# B&R Automation Studio project Panasonic_LinkaPowerCP2_A2021055 (part 8)

#### SKTcpClientTrace.c - SKTcpClientTrace
```c
/*************************************************************
*
*         projekt: SKTcp - Panasonic
*
*         autor: Ing. Milan Jun
*         company: B+R Automatizace spol. s r.o.
*         date: 10.09.2020
*
*/

#include <bur/plctypes.h>
#ifdef __cplusplus
	extern "C"
	{
#endif
#include "SKTcp.h"
#ifdef __cplusplus
	};
#endif

/* SKTcpClientTrace */
void SKTcpClientTrace(struct SKTcpClientTrace* inst)
{

	if( inst->Enable == 1 ) {

		if(( inst->Cmd.Send == 1 ) && ( inst->Internal.SendOld == 0 )) {
			inst->Internal.cmdSend = 1 ;
		}
		inst->Internal.SendOld = inst->Cmd.Send ;

		if(( inst->Cmd.Close == 1 ) && ( inst->Internal.CloseOld == 0 )) {
			inst->Internal.cmdClose = 1 ;
		} else {
			if( inst->Cmd.Close == 0 ) {
				inst->Internal.cmdClose = 0 ;
			}
		}
		inst->Internal.CloseOld = inst->Cmd.Close ;

		inst->Status.staSending = 0 ;
		inst->Status.staReceiving = 0 ;
		inst->Status.staReadyToSend = 0 ;
		inst->Status.staReadyToClose = 0 ;

		switch( inst->Internal.Step ) {

			case 0:
				inst->Status.staReadyToSend = 1 ;
				inst->Status.staSending = 0;
				inst->Internal.TimerIddle.IN = 0;

				if( inst->Internal.cmdSend == 1 ) {
					inst->FBStatus = 0xFFFF ;
					inst->Status.staSent = 0 ;
					inst->Status.staReceived = 0 ;

					inst->Status.staError = 0 ;
					inst->Status.staErrorSent = 0 ;
					inst->Status.staErrorOpen = 0 ;
					inst->Status.staErrorRecv = 0 ;
					inst->Status.staErrorRecvTout = 0 ;
					inst->Status.staErrorOpen = 0 ;
					inst->Status.staErrorIoctl = 0 ;
					inst->Status.staErrorClient = 0 ;
					inst->Status.staErrorConn = 0 ;
					inst->Status.staErrorConnTout = 0 ;

					inst->Status.RecvSize = 0 ;
					brsmemset((void*)&inst->Status.DataRecv[0], 0, sizeof(inst->Status.DataRecv)) ;

					inst->Internal.TimerConn.IN = 1 ;
					inst->Internal.TimerConn.PT = inst->Params.ConnTimeout ;

					inst->Internal.TCP_Open.enable = 1;
					inst->Internal.TCP_Open.pIfAddr = 0;
					inst->Internal.TCP_Open.port = inst->Params.IPportClient;
					inst->Internal.TCP_Open.options = 0;
					TcpOpen(&inst->Internal.TCP_Open);

					if( inst->Internal.TCP_Open.status == 0 ) {
						inst->Internal.Step = 4;
					}
					else if( inst->Internal.TimerConn.Q == 1 ) {
						inst->Internal.cmdSend = 0 ;
						inst->Status.staErrorOpen = 1 ;
						inst->Status.staErrorConn = 1 ;
						inst->Status.staErrorConnTout = 1 ;
						inst->Internal.Step = 99;
					} else if( inst->Internal.TCP_Open.status == ERR_FUB_BUSY ) {

					} else {
						if( inst->Internal.TCP_Open.status == tcpERR_ALREADY_EXIST ) {
							inst->Status.staErrorOpen = 1 ;
							inst->Internal.Step = 90;
						} else {
							inst->Status.staErrorOpen = 1 ;
							inst->Internal.Step = 99;
						}
						inst->Internal.cmdSend = 0 ;
					}
				}

				else if( inst->Cmd.Close == 1 ) {
					inst->Cmd.Close = 0 ;
					inst->Internal.Step = 40 ;
				}
				break ;

			case 4:
				inst->Internal.TimerIddle.IN = 1;
				inst->Internal.TimerIddle.PT = 1000;

				if( inst->Internal.TimerIddle.Q == 1 )
				{
					inst->Internal.TimerIddle.IN = 0 ;
					inst->Internal.Step = 5;
				}
				break ;

			case 5:
				inst->Internal.linger_opt.lLinger = 0;
				inst->Internal.linger_opt.lOnOff = 1;

				inst->Internal.TCP_Ioctl.enable = 1;
				inst->Internal.TCP_Ioctl.ident = inst->Internal.TCP_Open.ident;
				inst->Internal.TCP_Ioctl.ioctl = tcpSO_LINGER_SET;
				inst->Internal.TCP_Ioctl.pData = (UDINT)&(inst->Internal.linger_opt);
				inst->Internal.TCP_Ioctl.datalen = sizeof(inst->Internal.linger_opt);
				TcpIoctl(&inst->Internal.TCP_Ioctl);

				if( inst->Internal.TCP_Ioctl.status == 0 ) {
					inst->Internal.Step = 10;
				} else if( inst->Internal.TimerConn.Q == 1 ) {
					inst->Status.staErrorOpen = 1 ;
					inst->Status.staErrorConn = 1 ;
					inst->Status.staErrorConnTout = 1 ;
					inst->Internal.Step = 99;
				} else if( inst->Internal.TCP_Ioctl.status == ERR_FUB_BUSY ) {
				} else {
					inst->Status.staErrorIoctl = 1 ;
					inst->Internal.Step = 90;
				}
				break ;

			case 10:
				inst->Internal.TCP_Client.enable = 1;
				inst->Internal.TCP_Client.ident = inst->Internal.TCP_Open.ident ;
				inst->Internal.TCP_Client.portserv = inst->Params.IPportServ ;
				inst->Internal.TCP_Client.pServer = (UDINT)&inst->Params.IPaddrServ[0];
				TcpClient(&inst->Internal.TCP_Client) ;

				if( inst->Internal.TCP_Client.status == 0 ) {
					inst->Internal.Step = 15;
				} else if( inst->Internal.TimerConn.Q == 1 ) {
					inst->Status.staErrorOpen = 1 ;
					inst->Status.staErrorConn = 1 ;
					inst->Status.staErrorConnTout = 1 ;
					inst->Internal.Step = 90;
				} else if( inst->Internal.TCP_Client.status == ERR_FUB_BUSY ) {
				} else if( inst->Internal.TCP_Client.status == tcpERR_INVALID ) {
					inst->Status.staErrorClient = 1 ;
					inst->Status.staErrorConn = 1 ;
					inst->Internal.Step = 90;
				} else {
					inst->Status.staErrorClient = 1 ;
					inst->Internal.Step = 90;
				}
				break ;

			case 15:
				inst->Status.staReadyToSend = 1;
				inst->Status.staSending = 0;

				if ( inst->Internal.cmdSend == 1 ) {
					inst->Status.RecvSize = 0 ;
					inst->Internal.TimerRecv.IN = 0 ;
					inst->Internal.cmdSend = 0 ;
					brsmemset((void*)&inst->Status.DataRecv, 0, sizeof(inst->Status.DataRecv)) ;

					brsmemset((void*)&inst->Internal.Splitter.out, 0, sizeof(inst->Internal.Splitter.out));
					inst->Internal.Step = 18;
				}
				else if ( inst->Internal.cmdClose == 1 ) {
					inst->Internal.cmdClose=0;
					inst->Internal.Step = 40;
				}
				break ;

			case 18:

				inst->Status.staSending = 1;

				inst->Internal.oneskorenie.IN = 1;
				inst->Internal.oneskorenie.PT = 100; //ms  1000

				if ( inst->Internal.oneskorenie.Q == 1 ) {
					inst->Internal.oneskorenie.IN = 0;
					inst->Internal.Step = 19;
				}

				TON(&inst->Internal.oneskorenie);

				break ;

			case 19:

				inst->Params.Packet.internal.start = 0x02;
				inst->Params.Packet.internal.length_int = 0;
				//inst->Params.Packet.internal.xor = 0;
				inst->Params.Packet.internal.stop = 0x03;

				brsmemset((UDINT)&(inst->Params.Packet.internal.length_str), 0, sizeof(inst->Params.Packet.internal.length_str));
				brsmemset((UDINT)&(inst->Params.Packet.internal.xor_str), 0, sizeof(inst->Params.Packet.internal.xor_str));

				brsmemset((UDINT)&(inst->DataSend.send_data_a), 0, sizeof(inst->DataSend.send_data_a));
				brsstrcat((UDINT)&(inst->DataSend.send_data_a), (UDINT)&(inst->Params.Packet.type));
				brsstrcat((UDINT)&(inst->DataSend.send_data_a), (UDINT)&("|"));
				brsstrcat((UDINT)&(inst->DataSend.send_data_a), (UDINT)&(inst->Params.Packet.workplace));
				brsstrcat((UDINT)&(inst->DataSend.send_data_a), (UDINT)&("|"));
				brsstrcat((UDINT)&(inst->DataSend.send_data_a), (UDINT)&(inst->Params.Packet.rfid));
				brsstrcat((UDINT)&(inst->DataSend.send_data_a), (UDINT)&("|"));
				brsstrcat((UDINT)&(inst->DataSend.send_data_a), (UDINT)&(inst->Params.Packet.master));
				brsstrcat((UDINT)&(inst->DataSend.send_data_a), (UDINT)&("|"));
				brsstrcat((UDINT)&(inst->DataSend.send_data_a), (UDINT)&(inst->Params.Packet.dps1));
				brsstrcat((UDINT)&(inst->DataSend.send_data_a), (UDINT)&("|"));
				brsstrcat((UDINT)&(inst->DataSend.send_data_a), (UDINT)&(inst->Params.Packet.dps2));
				brsstrcat((UDINT)&(inst->DataSend.send_data_a), (UDINT)&("|"));
				brsstrcat((UDINT)&(inst->DataSend.send_data_a), (UDINT)&(inst->Params.Packet.dps3));
				brsstrcat((UDINT)&(inst->DataSend.send_data_a), (UDINT)&("|"));
				brsstrcat((UDINT)&(inst->DataSend.send_data_a), (UDINT)&(inst->Params.Packet.dps4));
				brsstrcat((UDINT)&(inst->DataSend.send_data_a), (UDINT)&("|"));
				brsstrcat((UDINT)&(inst->DataSend.send_data_a), (UDINT)&(inst->Params.Packet.dps5));
				brsstrcat((UDINT)&(inst->DataSend.send_data_a), (UDINT)&("|"));
				brsstrcat((UDINT)&(inst->DataSend.send_data_a), (UDINT)&(inst->Params.Packet.operator_id));
				brsstrcat((UDINT)&(inst->DataSend.send_data_a), (UDINT)&("|"));
				brsstrcat((UDINT)&(inst->DataSend.send_data_a), (UDINT)&(inst->Params.Packet.data_report));
				brsstrcat((UDINT)&(inst->DataSend.send_data_a), (UDINT)&("|"));
				brsstrcat((UDINT)&(inst->DataSend.send_data_a), (UDINT)&(inst->Params.Packet.result));

				inst->Params.Packet.internal.length_int = brsstrlen((UDINT)&inst->DataSend.send_data_a);

				inst->Params.Packet.internal.length_b_int = inst->Params.Packet.internal.length_int + SKTcpClientNod(inst->Params.Packet.internal.length_int);

				brsitoa(inst->Params.Packet.internal.length_b_int,(UDINT)&(inst->Params.Packet.internal.length_str));

				brsmemset((UDINT)&(inst->DataSend.send_data_b), 0, sizeof(inst->DataSend.send_data_b));
				brsstrcat((UDINT)&(inst->DataSend.send_data_b), (UDINT)&(inst->Params.Packet.internal.length_str));
				brsstrcat((UDINT)&(inst->DataSend.send_data_b), (UDINT)&("|"));
				brsstrcat((UDINT)&(inst->DataSend.send_data_b), (UDINT)&(inst->Params.Packet.type));
				brsstrcat((UDINT)&(inst->DataSend.send_data_b), (UDINT)&("|"));
				brsstrcat((UDINT)&(inst->DataSend.send_data_b), (UDINT)&(inst->Params.Packet.workplace));
				brsstrcat((UDINT)&(inst->DataSend.send_data_b), (UDINT)&("|"));
				brsstrcat((UDINT)&(inst->DataSend.send_data_b), (UDINT)&(inst->Params.Packet.rfid));
				brsstrcat((UDINT)&(inst->DataSend.send_data_b), (UDINT)&("|"));
				brsstrcat((UDINT)&(inst->DataSend.send_data_b), (UDINT)&(inst->Params.Packet.master));
				brsstrcat((UDINT)&(inst->DataSend.send_data_b), (UDINT)&("|"));
				brsstrcat((UDINT)&(inst->DataSend.send_data_b), (UDINT)&(inst->Params.Packet.dps1));
				brsstrcat((UDINT)&(inst->DataSend.send_data_b), (UDINT)&("|"));
				brsstrcat((UDINT)&(inst->DataSend.send_data_b), (UDINT)&(inst->Params.Packet.dps2));
				brsstrcat((UDINT)&(inst->DataSend.send_data_b), (UDINT)&("|"));
				brsstrcat((UDINT)&(inst->DataSend.send_data_b), (UDINT)&(inst->Params.Packet.dps3));
				brsstrcat((UDINT)&(inst->DataSend.send_data_b), (UDINT)&("|"));
				brsstrcat((UDINT)&(inst->DataSend.send_data_b), (UDINT)&(inst->Params.Packet.dps4));
				brsstrcat((UDINT)&(inst->DataSend.send_data_b), (UDINT)&("|"));
				brsstrcat((UDINT)&(inst->DataSend.send_data_b), (UDINT)&(inst->Params.Packet.dps5));
				brsstrcat((UDINT)&(inst->DataSend.send_data_b), (UDINT)&("|"));
				brsstrcat((UDINT)&(inst->DataSend.send_data_b), (UDINT)&(inst->Params.Packet.operator_id));
				brsstrcat((UDINT)&(inst->DataSend.send_data_b), (UDINT)&("|"));
				brsstrcat((UDINT)&(inst->DataSend.send_data_b), (UDINT)&(inst->Params.Packet.data_report));
				brsstrcat((UDINT)&(inst->DataSend.send_data_b), (UDINT)&("|"));
				brsstrcat((UDINT)&(inst->DataSend.send_data_b), (UDINT)&(inst->Params.Packet.result));
				brsstrcat((UDINT)&(inst->DataSend.send_data_b), (UDINT)&("|"));

				//inst->Params.Packet.internal.xor_str = SKTcpClientXor(inst->DataSend.send_data_b,inst->Params.Packet.internal.length_int);

				//SKTcpClientNod(inst->Params.Packet.internal.length_int);
				inst->Params.Packet.internal.xor_str = SKTcpClientXor(inst->DataSend.send_data_b, inst->Params.Packet.internal.length_b_int+2);

				brsmemset((UDINT)&(inst->DataSend.DataSend), 0, sizeof(inst->DataSend.DataSend));
				inst->DataSend.DataSend[0] = inst->Params.Packet.internal.start;
				brsstrcat((UDINT)&(inst->DataSend.DataSend), (UDINT)&(inst->Params.Packet.internal.length_str));
				brsstrcat((UDINT)&(inst->DataSend.DataSend), (UDINT)&("|"));
				brsstrcat((UDINT)&(inst->DataSend.DataSend), (UDINT)&(inst->Params.Packet.type));
				brsstrcat((UDINT)&(inst->DataSend.DataSend), (UDINT)&("|"));
				brsstrcat((UDINT)&(inst->DataSend.DataSend), (UDINT)&(inst->Params.Packet.workplace));
				brsstrcat((UDINT)&(inst->DataSend.DataSend), (UDINT)&("|"));
				brsstrcat((UDINT)&(inst->DataSend.DataSend), (UDINT)&(inst->Params.Packet.rfid));
				brsstrcat((UDINT)&(inst->DataSend.DataSend), (UDINT)&("|"));
				brsstrcat((UDINT)&(inst->DataSend.DataSend), (UDINT)&(inst->Params.Packet.master));
				brsstrcat((UDINT)&(inst->DataSend.DataSend), (UDINT)&("|"));
				brsstrcat((UDINT)&(inst->DataSend.DataSend), (UDINT)&(inst->Params.Packet.dps1));
				brsstrcat((UDINT)&(inst->DataSend.DataSend), (UDINT)&("|"));
				brsstrcat((UDINT)&(inst->DataSend.DataSend), (UDINT)&(inst->Params.Packet.dps2));
				brsstrcat((UDINT)&(inst->DataSend.DataSend), (UDINT)&("|"));
				brsstrcat((UDINT)&(inst->DataSend.DataSend), (UDINT)&(inst->Params.Packet.dps3));
				brsstrcat((UDINT)&(inst->DataSend.DataSend), (UDINT)&("|"));
				brsstrcat((UDINT)&(inst->DataSend.DataSend), (UDINT)&(inst->Params.Packet.dps4));
				brsstrcat((UDINT)&(inst->DataSend.DataSend), (UDINT)&("|"));
				brsstrcat((UDINT)&(inst->DataSend.DataSend), (UDINT)&(inst->Params.Packet.dps5));
				brsstrcat((UDINT)&(inst->DataSend.DataSend), (UDINT)&("|"));
				brsstrcat((UDINT)&(inst->DataSend.DataSend), (UDINT)&(inst->Params.Packet.operator_id));
				brsstrcat((UDINT)&(inst->DataSend.DataSend), (UDINT)&("|"));
				brsstrcat((UDINT)&(inst->DataSend.DataSend), (UDINT)&(inst->Params.Packet.data_report));
				brsstrcat((UDINT)&(inst->DataSend.DataSend), (UDINT)&("|"));
				brsstrcat((UDINT)&(inst->DataSend.DataSend), (UDINT)&(inst->Params.Packet.result));
				brsstrcat((UDINT)&(inst->DataSend.DataSend), (UDINT)&("|"));

				inst->Params.Packet.internal.ret_len = strlen((UDINT)&inst->DataSend.DataSend);

				if ( inst->Params.Packet.internal.xor_str != 0 ) {
					brsstrcat((UDINT)&(inst->DataSend.DataSend), (UDINT)&(inst->Params.Packet.internal.xor_str));
				}
				else {
					inst->DataSend.DataSend[inst->Params.Packet.internal.ret_len] = 0x00;
					inst->DataSend.DataSend[inst->Params.Packet.internal.ret_len+1] = 0x03;
				/*brsstrcat((UDINT)&(inst->DataSend.DataSend), (UDINT)&("\0"));*/

				}
				inst->Internal.Step = 20;

				break;

			case 20:

				inst->Status.staSending = 1 ;
				inst->Status.staSent = 0 ;

				inst->Internal.Splitter.enable = 0;

				inst->Internal.TCP_Send.enable = 1;
				inst->Internal.TCP_Send.ident = inst->Internal.TCP_Open.ident;
				inst->Internal.TCP_Send.pData = (UDINT)&inst->DataSend.DataSend;
				inst->Internal.TCP_Send.datalen = brsstrlen((UDINT)&inst->DataSend.DataSend) +5;
				inst->Internal.TCP_Send.flags = 0;
				TcpSend(&inst->Internal.TCP_Send);

				if( inst->Internal.TCP_Send.status == 0 ) {
					inst->Status.staSent = 1 ;
					if( inst->Params.disRecv == 0 ) {
						inst->Internal.TimerRecv.IN = 0 ;
						brsstrcat( (UDINT)&inst->DataSend.DataSend, (UDINT)&("\r\n") );
						inst->Internal.Step = 21;
					}
				} else if( inst->Internal.TCP_Send.status == ERR_FUB_BUSY )	{
					//				} else if (( inst->Internal.TCP_Send.status == tcpERR_SENTLEN ) || ( inst->Internal.TCP_Send.status == tcpERR_NOT_CONNECTED )) {
					//					inst->Internal.Step = 40;
				} else {
					inst->Status.staErrorSent = 1 ;
					inst->Internal.Step = 40;
				}
				break;

			case 21:

				if ( inst->Cmd.LoggerOn == 1 ) {

					inst->Internal.SKTcpLogger.enable=1;
					inst->Internal.SKTcpLogger.trigger=1;
					inst->Internal.SKTcpLogger.mode=0;
					inst->Internal.SKTcpLogger.pDevice=inst->pDevice;
					inst->Internal.SKTcpLogger.pFile=inst->pFile;
					inst->Internal.SKTcpLogger.pSrc=(UDINT)&inst->DataSend.DataSend;

					if ( inst->Internal.SKTcpLogger.active == 1 && inst->Internal.SKTcpLogger.done == 1 )
					{
						inst->Internal.SKTcpLogger.enable=0;
						inst->Internal.SKTcpLogger.trigger=0;
						inst->Internal.SKTcpLogger.mode=0;
						inst->Internal.Step = 30;
					}
				}
				else if ( inst->Cmd.LoggerOn == 0 ) {
					inst->Internal.Step = 30;
				}

				break;

			case 30:

				inst->Status.staReceiving = 1 ;
				inst->Status.staReceived = 0 ;

				inst->Internal.TimerRecv.IN = 1 ;
				inst->Internal.TimerRecv.PT = inst->Params.RecvTimeout ;

				inst->Internal.TCP_Recv.enable = 1;
				inst->Internal.TCP_Recv.ident = inst->Internal.TCP_Open.ident;
				inst->Internal.TCP_Recv.pData	= (UDINT)&inst->Status.DataRecv;
				inst->Internal.TCP_Recv.datamax = sizeof(inst->Status.DataRecv);
				inst->Internal.TCP_Recv.flags = 0;
				TcpRecv(&inst->Internal.TCP_Recv);

				if( inst->Internal.TCP_Recv.status == 0 ) {
					inst->Status.staReceived = 1 ;
					inst->Status.RecvSize = inst->Internal.TCP_Recv.recvlen;
					inst->Status.RecvCounter++ ;

					brsmemcpy((UDINT)&inst->Internal.Splitter.iSelector,(UDINT)&("|"),sizeof("|"));
					brsmemcpy((UDINT)&inst->Internal.Splitter.iInputString,(UDINT)&(inst->Status.DataRecv),sizeof(inst->Status.DataRecv));
					inst->Internal.Splitter.enable = 1;

					if( inst->Params.enaClose == 1 ) {
						inst->Internal.TimerRecv.IN = 0 ;
						inst->Internal.Step = 40;
					} else {
						inst->Internal.TimerRecv.IN = 0 ;
						brsstrcat( (UDINT)&inst->Status.DataRecv, (UDINT)&("\r\n") );
						inst->Internal.Step = 31;
					}

				}
				else if( inst->Internal.TCP_Recv.status == tcpERR_NO_DATA ) {
					if( inst->Internal.TimerRecv.Q == 1 ) {
						inst->Status.staErrorRecvTout = 1 ;
						inst->Internal.TimerRecv.IN = 0 ;
						inst->Internal.Step = 40;
					}
				}
				else if ( inst->Internal.TCP_Recv.status == ERR_FUB_BUSY ) {

				}
				else if( inst->Internal.TCP_Recv.status == tcpERR_NOT_CONNECTED ) {
					inst->Status.staErrorRecv = 1 ;
					inst->Internal.TimerRecv.IN = 0 ;
					inst->Internal.Step = 40;
				}

				if( inst->Internal.TimerRecv.Q == 1 ) {
					inst->Status.staErrorRecv = 1 ;
					inst->Internal.TimerRecv.IN = 0 ;
					inst->Internal.Step = 40;
				}

				if ( inst->Internal.cmdClose == 1 ) {
					inst->Internal.cmdClose=0;
					inst->Internal.TimerRecv.IN = 0 ;
					inst->Internal.Step = 40;
				}

				break ;

			case 31:

				if ( inst->Cmd.LoggerOn == 1 ) {
					inst->Internal.SKTcpLogger.enable=1;
					inst->Internal.SKTcpLogger.trigger=1;
					inst->Internal.SKTcpLogger.mode=1;
					inst->Internal.SKTcpLogger.pDevice=inst->pDevice;
					inst->Internal.SKTcpLogger.pFile=inst->pFile;
					inst->Internal.SKTcpLogger.pSrc=(UDINT)&inst->Status.DataRecv;

					if ( inst->Internal.SKTcpLogger.active == 1 && inst->Internal.SKTcpLogger.done == 1 )
					{
						inst->Internal.SKTcpLogger.enable=0;
						inst->Internal.SKTcpLogger.trigger=0;
						inst->Internal.SKTcpLogger.mode=0;
						inst->Internal.Step = 15;
					}
				}
				else if ( inst->Cmd.LoggerOn == 0 ) {
					inst->Internal.Step = 15;
				}

				break;

			case 40:
				inst->Internal.TCP_Open.enable = 0;
				inst->Status.staReadyToSend = 0;
				inst->Internal.TCP_Close.enable = 1;
				inst->Internal.TCP_Close.ident = inst->Internal.TCP_Open.ident ;
				inst->Internal.TCP_Close.how = 0;
				TcpClose(&inst->Internal.TCP_Close);

				if( inst->Internal.TCP_Close.status == 0 ) {
					inst->Internal.Step = 100;
					inst->Status.staReceived = 1 ;
				} else if( inst->Internal.TCP_Close.status == ERR_FUB_BUSY ) {
				} else {
					inst->Status.staErrorClose = 1 ;
					inst->Internal.Step = 99;
				}
				break ;

			case 90:
				inst->Internal.TCP_Close.enable = 1;
				inst->Internal.TCP_Close.ident = inst->Internal.TCP_Open.ident;
				inst->Internal.TCP_Close.how = 0;
				TcpClose(&inst->Internal.TCP_Close);

				if( inst->Internal.TCP_Close.status == 0 ) {
					inst->Internal.Step = 99;
				} else if( inst->Internal.TCP_Close.status == ERR_FUB_BUSY ) {
				} else {
					inst->Status.staErrorClose = 1 ;
					inst->Internal.Step = 99;
				}
				break ;

			case 99:

				inst->FBStatus = 1 ;
				inst->Status.staError = 1 ; ;
				inst->Internal.Step = 0;
				inst->Internal.TimerConn.IN = 0 ;
				inst->Internal.cmdSend = 0 ;

				break ;

			case 100:
				inst->FBStatus = 0 ;
				inst->Internal.Step = 0;
				inst->Internal.cmdSend = 0 ;
				inst->Internal.TimerConn.IN = 0 ;
				break ;

		}

		SKTcpLogger(&inst->Internal.SKTcpLogger);

	} else {
		if( inst->Cmd.Send == 0 ) {
			inst->FBStatus = 0xFFFE ;
		}

		if( inst->Internal.TCP_Open.ident != 0 ) {
			inst->Internal.TCP_Close.enable = 1;
			inst->Internal.TCP_Close.ident = inst->Internal.TCP_Open.ident;
			inst->Internal.TCP_Close.how = 0;
			TcpClose(&inst->Internal.TCP_Close);

			if( inst->Internal.TCP_Close.status == 0 ) {
			} else if( inst->Internal.TCP_Close.status == ERR_FUB_BUSY ) {
			} else {
			}
		}
		inst->Internal.TimerRecv.IN = 0 ;
		inst->Internal.TimerConn.IN = 0 ;
		inst->Internal.Step = 0 ;
	}

	inst->Internal.EnableOld = inst->Enable ;
	TON(&inst->Internal.TimerRecv) ;
	TON(&inst->Internal.TimerConn) ;
	TON(&inst->Internal.TimerIddle) ;
	SKTcpClientSplitter(&inst->Internal.Splitter);

}
```

#### SKTcpClientSplitter.c - SKTcpClientSplitter
```c
/*************************************************************
*
*         projekt: SKTcp - Panasonic
*
*         autor: Ing. Milan Jun
*         company: B+R Automatizace spol. s r.o.
*         date: 10.09.2020
*
*/

#include <bur/plctypes.h>
#ifdef __cplusplus
	extern "C"
	{
#endif
#include "SKTcp.h"
#ifdef __cplusplus
	};
#endif

/* SKTcpClientSplitter */
void SKTcpClientSplitter(struct SKTcpClientSplitter* inst)
{

	if ( inst->enable == 0 )
	{

		inst->done = 0;

		brsmemset((UDINT)&(inst->out), 0, sizeof(inst->out));
		brsmemset((UDINT)&(inst->OUT_Master), 0, sizeof(inst->OUT_Master));
		brsmemset((UDINT)&(inst->OUT_Typ), 0, sizeof(inst->OUT_Typ));
		brsmemset((UDINT)&(inst->OUT_Result), 0, sizeof(inst->OUT_Result));
		brsmemset((UDINT)&(inst->tmpInputString), 0, sizeof(inst->tmpInputString));
		brsmemset((UDINT)&(inst->tmpString), 0, sizeof(inst->tmpString));
		brsmemset((UDINT)&(inst->idx), 0, sizeof(inst->idx));

	}
	else if ( inst->enable == 1 )
	{

		if ( inst->enable == 1 && inst->enableOld==0 )
		{
			inst->enableOld = 1;

			brsmemcpy ((UDINT)&(inst->tmpInputString),(UDINT)&(inst->iInputString), brsstrlen((UDINT)&(inst->iInputString)));

			inst->idx[1] = 0;

			if ( strlen((UDINT)&(inst->iInputString)) != 0 )
			{

				for (inst->idx[0] = 0; inst->idx[0] < brsstrlen(inst->iInputString) ; inst->idx[0]++)
				{

					if ( inst->iSelector != inst->tmpInputString[inst->idx[0]] )
					{
						brsmemcpy((UDINT)&(inst->tmpString),(UDINT)&(inst->tmpInputString[inst->idx[0]]),1);
						brsstrcat((UDINT)&(inst->out[inst->idx[1]]),(UDINT)&(inst->tmpString));

					}
					else
					{
						inst->idx[1]++;
					}

				}
				brsmemcpy((UDINT)&(inst->OUT_Master),(UDINT)&(inst->out[4]),30);
				brsmemcpy((UDINT)&(inst->OUT_Typ),(UDINT)&(inst->out[1]),1);
				brsmemcpy((UDINT)&(inst->OUT_Result),(UDINT)&(inst->out[12]),2);
			}

		}

	}

	inst->enableOld = inst->enable;

}
```

#### SKTcpClientXor.c - SKTcpClientXor
```c
/*************************************************************
*
*         projekt: SKTcp - Panasonic
*
*         autor: Ing. Milan Jun
*         company: B+R Automatizace spol. s r.o.
*         date: 10.09.2020
*
*/

#include <bur/plctypes.h>
#ifdef __cplusplus
	extern "C"
	{
#endif
#include "SKTcp.h"
#ifdef __cplusplus
	};
#endif

/* SKTcpClientXor */
unsigned char SKTcpClientXor(unsigned char in[MAX_STRING_MINUS_ONE], unsigned short len)
{

	unsigned char xor_byte = 0;
	unsigned short tI = 0;

	for (tI = 0; tI < len; tI++) xor_byte = xor_byte ^ in[tI];

	return xor_byte;

}
```

#### SKTcpClientNod.c - SKTcpClientNod
```c
/*************************************************************
*
*         projekt: SKTcp - Panasonic
*
*         autor: Ing. Milan Jun
*         company: B+R Automatizace spol. s r.o.
*         date: 10.09.2020
*
*/

#include <bur/plctypes.h>
#ifdef __cplusplus
	extern "C"
	{
#endif
#include "SKTcp.h"
#ifdef __cplusplus
	};
#endif

/* SKTcpClientNod */
unsigned short SKTcpClientNod(unsigned long n)
{

	unsigned int count = 0;

	while (n != 0) { n /= 10; ++count; }

	return count;

}
```

#### SKTcpClientEdge.c - SKTcpClientEdge
```c
/*************************************************************
*
*         projekt: SKTcp - Panasonic
*
*         autor: Ing. Milan Jun
*         company: B+R Automatizace spol. s r.o.
*         date: 10.09.2020
*
*/

#include <bur/plctypes.h>
#ifdef __cplusplus
	extern "C"
	{
#endif
#include "SKTcp.h"
#ifdef __cplusplus
	};
#endif

/* SKTcpClientEdge */
void SKTcpClientEdge(struct SKTcpClientEdge* inst)
{

	inst->Q = ( ! inst->CLK == inst->Last_State) ;

	inst->Last_State = inst->CLK;

}
```

#### SKTcpClientNewCsvEntry.c - SKTcpClientNewCsvEntry
```c
/*************************************************************
*
*         projekt: SKTcp - Panasonic
*
*         autor: Ing. Milan Jun
*         company: B+R Automatizace spol. s r.o.
*         date: 21.09.2020
*
*/

#include <bur/plctypes.h>
#ifdef __cplusplus
	extern "C"
	{
#endif
#include "SKTcp.h"
#ifdef __cplusplus
	};
#endif

/* SKTcpClientNewCsvEntry */
unsigned char SKTcpClientNewCsvEntry(plcstring* IDstep, plcstring* Description, plcstring* TypeValue, plcstring* MinTol, plcstring* MaxTol, plcstring* Nom, plcstring* MinEle, plcstring* MaxEle, plcstring* Value, plcstring* ValEle, plcstring* Result, unsigned long pData)
{

	/* SKTcpClientNewCsvEntry('IDstep','Description','TypeValue','MinTol','MaxTol','Nom','MinEle','MaxEle','Value','ValEle','Result', ADR(CSV)); */

	brsstrcat((void*)pData, IDstep);
	brsstrcat((void*)pData, (UDINT)&";");
	brsstrcat((void*)pData, Description);
	brsstrcat((void*)pData, (UDINT)&";");
	brsstrcat((void*)pData, TypeValue);
	brsstrcat((void*)pData, (UDINT)&";");
	brsstrcat((void*)pData, MinTol);
	brsstrcat((void*)pData, (UDINT)&";");
	brsstrcat((void*)pData, MaxTol);
	brsstrcat((void*)pData, (UDINT)&";");
	brsstrcat((void*)pData, Nom);
	brsstrcat((void*)pData, (UDINT)&";");
	brsstrcat((void*)pData, MinEle);
	brsstrcat((void*)pData, (UDINT)&";");
	brsstrcat((void*)pData, MaxEle);
	brsstrcat((void*)pData, (UDINT)&";");
	brsstrcat((void*)pData, Value);
	brsstrcat((void*)pData, (UDINT)&";");
	brsstrcat((void*)pData, ValEle);
	brsstrcat((void*)pData, (UDINT)&";");
	brsstrcat((void*)pData, Result);
	brsstrcat((void*)pData, (UDINT)&("\r"));

	return 0;
}
```

#### SKTcpClientNewLoggerEntry.c - SKTcpClientNewLoggerEntry
```c
/*************************************************************
*
*         projekt: SKTcp - Panasonic
*
*         autor: Ing. Milan Jun
*         company: B+R Automatizace spol. s r.o.
*         date: 21.09.2020
*
*/

#include <bur/plctypes.h>
#ifdef __cplusplus
	extern "C"
	{
#endif
#include "SKTcp.h"
#ifdef __cplusplus
	};
#endif

/* SKTcpClientNewLoggerEntry */
unsigned char SKTcpClientNewLoggerEntry(plcstring* msg, UDINT pData, UINT entrys)
{

	RTCtime_typ	RTCtime_struct;
	STRING lstr1[5000], lstr2[5000];

	if ((entrys > 0) && (pData != 0))
	{
		brsstrcpy(lstr1, "");
		brsstrcpy(lstr2, "");
		RTC_gettime(&RTCtime_struct);
		brsitoa(RTCtime_struct.hour, (UDINT)&lstr1);
		if(brsstrlen(lstr1) == 1) brsstrcat(lstr2, "0");
		brsstrcat(lstr2, lstr1);
		brsstrcat(lstr2, ":");
		brsitoa(RTCtime_struct.minute, (UDINT)&lstr1);
		if(brsstrlen(lstr1) == 1) brsstrcat(lstr2, "0");
		brsstrcat(lstr2, lstr1);
		brsstrcat(lstr2, ":");
		brsitoa(RTCtime_struct.second, (UDINT)&lstr1);
		if(brsstrlen(lstr1) == 1) brsstrcat(lstr2, "0");
		brsstrcat(lstr2, lstr1);
		brsstrcat(lstr2, ":");
		brsitoa(RTCtime_struct.millisec, (UDINT)&lstr1);
		if(brsstrlen(lstr1) == 1) brsstrcat(lstr2, "00");
		if(brsstrlen(lstr1) == 2) brsstrcat(lstr2, "0");
		brsstrcat(lstr2, lstr1);
		brsstrcat(lstr2, " ");
		brsstrcat(lstr2, msg);
		brsmemmove((void*)(pData)+5001, (void*)pData, 5001*(entrys-1));
		brsstrcpy((void*)pData, lstr2);
	}

	return 0;

}
```

#### SKTcpClientSC.c - SKTcpClientSC
```c
/*************************************************************
*
*         projekt: SKTcp - Panasonic
*
*         autor: Ing. Milan Jun
*         company: B+R Automatizace spol. s r.o.
*         date: 21.09.2020
*
*/

#include <bur/plctypes.h>
#ifdef __cplusplus
	extern "C"
	{
#endif
#include "SKTcp.h"
#ifdef __cplusplus
	};
#endif

/* SKTcpClientSC */
unsigned char SKTcpClientSC(struct SKTcpClientSC_Type* sc)
{

	if ( sc->bNext == 1 ) {

		sc->bNext = 0;
		sc->bRepeat = 0;
		sc->edge = 0;
		sc->step++;

	}

	if ( sc->bLast == 1 ) {

		sc->bLast = 0;
		sc->bRepeat = 0;
		sc->edge = 0;
		sc->step = 0;

	}

	if ( sc->bJump == 1 ) {

		sc->bJump = 0;
		sc->bRepeat = 0;
		sc->edge = 0;

	}

	TON(&sc->idle_time);
	TON(&sc->alarm_time);

	return 0;

}
```

#### SKTcpLogger.c - SKTcpLogger
```c
#include <bur/plctypes.h>
#ifdef __cplusplus
	extern "C"
	{
#endif
#include "SKTcp.h"
#include <AsBrStr.h>
#include <sys_lib.h>
#ifdef __cplusplus
	};
#endif

void SKTcpLogger(struct SKTcpLogger* inst)
{

	RTCtime_typ	RTCtime_struct;
	STRING		lstr1[5000], lstr2[5000];

	if ( inst->enable == 1 )
	{
		switch ( inst->internal.step )
		{
			case 0:

				if ( inst->trigger == 1 )
					inst->internal.step++;

				break;

			case 1:
				inst->internal.FileOpen.enable = 1;
				inst->internal.FileOpen.pDevice = inst->pDevice;
				inst->internal.FileOpen.pFile = inst->pFile;
				inst->internal.FileOpen.mode = fiREAD_WRITE;
				FileOpen(&inst->internal.FileOpen);
				if ( inst->internal.FileOpen.status == ERR_OK ) {
					inst->internal.FileOpen.enable = 0;
					inst->internal.step++;
				}
				break;

			case 2:

				brsstrcpy(lstr1, "");
				brsstrcpy(lstr2, "");

				RTC_gettime(&RTCtime_struct);

				brsitoa(RTCtime_struct.year, (UDINT)&lstr1);
				if(brsstrlen(lstr1) == 1) brsstrcat(lstr2, "0");
				brsstrcat(lstr2, lstr1);
				brsstrcat(lstr2, "-");
				brsitoa(RTCtime_struct.month, (UDINT)&lstr1);
				if(brsstrlen(lstr1) == 1) brsstrcat(lstr2, "0");
				brsstrcat(lstr2, lstr1);
				brsstrcat(lstr2, "-");
				brsitoa(RTCtime_struct.day, (UDINT)&lstr1);
				if(brsstrlen(lstr1) == 1) brsstrcat(lstr2, "0");
				brsstrcat(lstr2, lstr1);
				brsstrcat(lstr2, " ");
				brsitoa(RTCtime_struct.hour, (UDINT)&lstr1);
				if(brsstrlen(lstr1) == 1) brsstrcat(lstr2, "0");
				brsstrcat(lstr2, lstr1);
				brsstrcat(lstr2, ":");
				brsitoa(RTCtime_struct.minute, (UDINT)&lstr1);
				if(brsstrlen(lstr1) == 1) brsstrcat(lstr2, "0");
				brsstrcat(lstr2, lstr1);
				brsstrcat(lstr2, ":");
				brsitoa(RTCtime_struct.second, (UDINT)&lstr1);
				if(brsstrlen(lstr1) == 1) brsstrcat(lstr2, "0");
				brsstrcat(lstr2, lstr1);
				brsstrcat(lstr2, ":");
				brsitoa(RTCtime_struct.millisec, (UDINT)&lstr1);
				if(brsstrlen(lstr1) == 1) brsstrcat(lstr2, "00");
				if(brsstrlen(lstr1) == 2) brsstrcat(lstr2, "0");
				brsstrcat(lstr2, lstr1);

				brsstrcat(lstr2, " ");

				if ( inst->mode == 0 )
					brsstrcat(lstr2, " -> ");

				if ( inst->mode == 1 )
					brsstrcat(lstr2, " <- ");

				brsstrcat(lstr2, " ");

				brsstrcpy((UDINT)&inst->internal.data, lstr2);
				brsstrcat((UDINT)&inst->internal.data, inst->pSrc);
				brsstrcat((UDINT)&inst->internal.data, (UDINT)&"\r");

				inst->internal.step++;
				break;

			case 3:
				inst->internal.FileWrite.enable = 1;
				inst->internal.FileWrite.ident = inst->internal.FileOpen.ident;
				inst->internal.FileWrite.offset = inst->internal.FileOpen.filelen;
				inst->internal.FileWrite.pSrc = (UDINT)&inst->internal.data;
				inst->internal.FileWrite.len = brsstrlen((UDINT)&inst->internal.data);
				FileWrite(&inst->internal.FileWrite);
				if ( inst->internal.FileWrite.status == ERR_OK ) {
					inst->internal.FileWrite.enable = 0;
					inst->internal.step++;
				}
				break;

			case 4:
				inst->internal.FileClose.enable = 1;
				inst->internal.FileClose.ident = inst->internal.FileOpen.ident;
				FileClose(&inst->internal.FileClose);
				if ( inst->internal.FileClose.status == ERR_OK ) {
					inst->internal.FileClose.enable = 0;
					inst->internal.step++;
				}
				break;

			case 5:
				inst->done = 1;
				break;
		}

		inst->active = 1;

		if ( inst->trigger == 0 )
		{
			inst->internal.step = 0;
			inst->done = 0;
		}

	}
	else if ( inst->enable == 0 )
	{
		inst->internal.step = 0;
		inst->active = 0;
		inst->done = 0;
	}
}
```

### Package Logical/Program - Riadiace programy

### Program Logical/Program/Linka/Main (IEC)

#### Main.st - Init, cyclic, exit code
```iecst
PROGRAM _INIT

	P3_LeakageTestA.STAV.Tester_ON:= TRUE;
	P3_LeakageTestB.STAV.Tester_ON:= TRUE;
	P4_FunkcnyTestA.STAV.Tester_ON:= TRUE;
	P4_FunkcnyTestB.STAV.Tester_ON:= TRUE;
	Linka.PAR.IndexModelu:= 1;
	Linka.KOM_FTP_OFF:= FALSE;
	Linka.KOM_Panatrace_OFF:= FALSE;
	Linka.P1_Kamery_OFF:= FALSE;
	Linka.P2_Kamery_OFF:= FALSE;
	Linka.P3_Kamery_OFF:= FALSE;
	Linka.P4_Kamery_OFF:= FALSE;
	Linka.P1_SkrutkovanieResult_OFF:= FALSE;
	Linka.P2_SkrutkovanieResult_OFF:= FALSE;
	Linka.P3_SkrutkovanieResult_OFF:= FALSE;
	P2_Vizu.ZobrazHL5_ST5:= FALSE;
	P2_Vizu.ZobrazHL6_ST5:= TRUE;
	P2_Vizu.ZobrazHL7_ST5:= FALSE;

END_PROGRAM

PROGRAM _CYCLIC

 //Volanie podprogramov//
ProfinetKomunikaciaCU;

	TypFotky_BMP;

	//**************************Zmena času a dátumu***************************************//
	IF Vizu.NastavCasPLC THEN
		DTSetTime_0.enable:= TRUE;
		DTSetTime_0.DT1:= Vizu.ZadanyCasPLC;
		DTSetTime_0();
	END_IF

	IF DTSetTime_0.status = 0 THEN
		Vizu.NastavCasPLC:= FALSE;
		DTSetTime_0.enable:= FALSE;
		DTSetTime_0();
	END_IF

	//**********************Načítanie času a dátumu do vizualizácie**************************//
	DTGetTime_0.enable:= TRUE;
	Vizu.AktualnyCasPLC:= DTGetTime_0.DT1;
	DTGetTime_0();

	//Volba modelu//
	IF Linka.STAV.OFF THEN
		IF Linka.PAR.IndexModelu = 0 THEN
			Linka.PAR.ZvolenyModel:= '4F';
		ELSIF Linka.PAR.IndexModelu = 1 THEN
			Linka.PAR.ZvolenyModel:= '5F';
		ELSIF Linka.PAR.IndexModelu = 2 THEN
			Linka.PAR.ZvolenyModel:= '5H';
		END_IF
	END_IF

	//**************************Stav linka vypnuta********************************************//
	IF P1_Pracovisko.STAV.Automat THEN
		Linka.STAV.OFF:= FALSE;
	ELSIF P2_Pracovisko.STAV.Automat THEN
		Linka.STAV.OFF:= FALSE;
	ELSIF P3_Pracovisko.STAV.Automat THEN
		Linka.STAV.OFF:= FALSE;
	ELSIF P4_Pracovisko.STAV.Automat THEN
		Linka.STAV.OFF:= FALSE;
	ELSE
		Linka.STAV.OFF:= TRUE;
	END_IF

	//**************************Stav linka prazdna********************************************//
	IF NOT P1_StoperSrobovania.RFID_hlava.PritomnostPaletky AND
		NOT P1_AkumulacnyStoper.IN.PritomnostPaletky AND
		NOT P2_StoperZaklTesnenia.RFID_hlava.PritomnostPaletky AND
		NOT P2_StoperMaticovacky.RFID_hlava.PritomnostPaletky AND
		NOT P2_AkumulacnyStoper.IN.PritomnostPaletky AND
		NOT P2_StoperSrobovania.RFID_hlava.PritomnostPaletky AND
		NOT P2_StoperZvarania.RFID_hlava.PritomnostPaletky AND
		NOT P3_StoperSrobovania.RFID_hlava.PritomnostPaletky AND
		NOT P3_HV_Test.RFID_hlava.PritomnostPaletky AND
		NOT P3_ZdvizkaPredLeakTestA.IN.PritomnostPaletky AND
		NOT P3_ZdvizkaPredLeakTestB.IN.PritomnostPaletky AND
		NOT P3_LeakageTestA.RFID_hlava.PritomnostPaletky AND
		NOT P3_LeakageTestB.RFID_hlava.PritomnostPaletky AND
		NOT P3_ZdvizkaZaLeakTestA.IN.PritomnostPaletky AND
		NOT P3_ZdvizkaZaLeakTestB.IN.PritomnostPaletky AND
		NOT P4_FunkcnyTestA.RFID_hlava.PritomnostPaletky AND
		NOT P4_FunkcnyTestB.RFID_hlava.PritomnostPaletky AND
		NOT P4_ZdvizkaZaFunkcTestA.IN.PritomnostPaletky AND
		NOT P4_ZdvizkaZaFunkcTestB.IN.PritomnostPaletky AND
		NOT P4_Etiketovacka.RFID_hlava.PritomnostPaletky AND
		NOT P4_Vytah.RFID_hlava.PritomnostPaletky THEN
		Linka.STAV.PRAZDNA:= TRUE;
	ELSE
		Linka.STAV.PRAZDNA:= FALSE;
	END_IF

	//***************************Stav linka po init********************************//

	IF P1_Pracovisko.STAV.PoINIT AND
		P2_Pracovisko.STAV.PoINIT AND
		P3_Pracovisko.STAV.PoINIT AND
		P4_Pracovisko.STAV.PoINIT THEN
		Linka.STAV.PoINIT:= TRUE;
	ELSE
		Linka.STAV.PoINIT:= FALSE;
	END_IF

END_PROGRAM

PROGRAM _EXIT
	(* Insert code here *)

END_PROGRAM
```

#### ProfinetKomunikaciaCU.st
```iecst
ACTION ProfinetKomunikaciaCU:

	//Stavy jednotky pre ovládanie kamier//
	ControlUnit.Stav_READY:= ControlUnit.Profinet_PLC_INPUTS[0].0;

END_ACTION
```

### Program Logical/Program/Linka/OvladanieSafety (IEC)

#### Main.st - Init, cyclic, exit code
```iecst
PROGRAM _INIT
	(* Insert code here *)

END_PROGRAM

PROGRAM _CYCLIC

	//*************************************Príznak tlačítka CS odblokované**********************************************//
	IF Safety.STAV.P1_Panel_TlacitkoCS_ODBLOK AND
		Safety.STAV.P1_Robot_TlacitkoCS_ODBLOK AND
		Safety.STAV.P1_Rozvadzac_TlacitkoCS_ODBLOK AND
		Safety.STAV.P2_Panel_TlacitkoCS_ODBLOK AND
		Safety.STAV.P2_DvojrucOvl_TlacitkoCS_ODBLOK AND
		Safety.STAV.P2_Robot_TlacitkoCS_ODBLOK AND
		Safety.STAV.P2_Rozvadzac_TlacitkoCS_ODBLOK AND
		Safety.STAV.P3_Rozvadzac_TlacitkoCS_ODBLOK AND
		Safety.STAV.P4_Panel_TlacitkoCS_ODBLOK AND
		Safety.STAV.P4_Rozvadzac_TlacitkoCS_ODBLOK THEN
		Safety.STAV.Linka_TlacitkaCS_ODBLOKOVANE:= TRUE;
	ELSE
		Safety.STAV.Linka_TlacitkaCS_ODBLOKOVANE:= FALSE;
	END_IF

	//******************************************Reset zóny CS*******************************************************//
	IF P1_Vizu.TL_ResetCS THEN
		Safety.OUT.Linka_ResetCS:= TRUE;
		P1_Vizu.TL_ResetCS:= FALSE;
	ELSIF P2_Vizu.TL_ResetCS THEN
		Safety.OUT.Linka_ResetCS:= TRUE;
		P2_Vizu.TL_ResetCS:= FALSE;
	ELSIF P34_Vizu.TL_ResetCS THEN
		Safety.OUT.Linka_ResetCS:= TRUE;
		P34_Vizu.TL_ResetCS:= FALSE;
	END_IF

	IF Safety.OUT.Linka_ResetCS THEN
		IF Safety.STAV.Linka_ZonaCS_AKTIVNA THEN
			Safety.OUT.Linka_ResetCS:= FALSE;
		ELSIF NOT Safety.STAV.Linka_TlacitkaCS_ODBLOKOVANE THEN
			Safety.OUT.Linka_ResetCS:= FALSE;
		END_IF
	END_IF

	//***************************************Príznak safety PLC nabehlo*********************************************//
    CasNabehnutiaSafetyPLC.PT:= T#10s;
	CasNabehnutiaSafetyPLC();

	CasNabehnutiaSafetyPLC.IN:= Linka.IN.SafetyMaster_OK;

	IF CasNabehnutiaSafetyPLC.Q THEN
		Safety.STAV.Linka_SafetyPLC_Nabehlo:= TRUE;
	ELSE
		Safety.STAV.Linka_SafetyPLC_Nabehlo:= FALSE;
	END_IF

END_PROGRAM

PROGRAM _EXIT
	(* Insert code here *)

END_PROGRAM
```

#### Variables.var - Local variables
```iecst
VAR
	CasNabehnutiaSafetyPLC : TON := (0);
END_VAR
```

### Program Logical/Program/Linka/OvladanieVizu (IEC)

#### Main.st - Init, cyclic, exit code
```iecst
PROGRAM _INIT
	(* Insert code here *)

END_PROGRAM

PROGRAM _CYCLIC

	//**************************************Zmena farby tlačítok Reset CS *********************************************//
	IF Safety.STAV.Linka_ZonaCS_AKTIVNA THEN
		Vizu.TL_ResetCS_Farba:= "Button_Green";
	ELSIF NOT Safety.STAV.Linka_ZonaCS_AKTIVNA AND Safety.STAV.Linka_TlacitkaCS_ODBLOKOVANE THEN
		IF Blikac1s THEN
			Vizu.TL_ResetCS_Farba:= "Button_Blue";
		ELSE
			Vizu.TL_ResetCS_Farba:= "Operate";
		END_IF
	ELSE
		Vizu.TL_ResetCS_Farba:= "Button_Red";
	END_IF

	//************************************Blokovanie tlačítok prihlásenia operátora*************************************//
	IF P1_Vizu.TL_PrihlasovOperatora_AKTIVNE THEN
		P2_Vizu.TL_PrihlasovOperatora_AKTIVNE:= FALSE;
		P34_Vizu.TL_PrihlasovOperatora_AKTIVNE:= FALSE;
		P2_Vizu.TL_PrihlasenieOperatora_ENABLE:= FALSE;
		P34_Vizu.TL_PrihlasenieOperatora_ENABLE:= FALSE;
	ELSIF P2_Vizu.TL_PrihlasovOperatora_AKTIVNE THEN
		P1_Vizu.TL_PrihlasovOperatora_AKTIVNE:= FALSE;
		P34_Vizu.TL_PrihlasovOperatora_AKTIVNE:= FALSE;
		P1_Vizu.TL_PrihlasenieOperatora_ENABLE:= FALSE;
		P34_Vizu.TL_PrihlasenieOperatora_ENABLE:= FALSE;
	ELSIF P34_Vizu.TL_PrihlasovOperatora_AKTIVNE THEN
		P1_Vizu.TL_PrihlasovOperatora_AKTIVNE:= FALSE;
		P2_Vizu.TL_PrihlasovOperatora_AKTIVNE:= FALSE;
		P1_Vizu.TL_PrihlasenieOperatora_ENABLE:= FALSE;
		P2_Vizu.TL_PrihlasenieOperatora_ENABLE:= FALSE;
	ELSE
		P1_Vizu.TL_PrihlasenieOperatora_ENABLE:= TRUE;
		P2_Vizu.TL_PrihlasenieOperatora_ENABLE:= TRUE;
		P34_Vizu.TL_PrihlasenieOperatora_ENABLE:= TRUE;
	END_IF

	//************************************Vypnutie tlačítok prihlásenie operátora*********************************************//
	//Panel 1//
	IF P1_UzivatelPrihlaseny AND P1_Vizu.TL_PrihlasovOperatora_AKTIVNE AND P1_Vizu.ActualPage <> 'PageUsers' THEN
		P1_Vizu.TL_PrihlasovOperatora_AKTIVNE:= FALSE;
	END_IF

	//Panel 2//
	IF P2_UzivatelPrihlaseny AND P2_Vizu.TL_PrihlasovOperatora_AKTIVNE THEN
		P2_Vizu.TL_PrihlasovOperatora_AKTIVNE:= FALSE;
	END_IF

	//Panel 3//
	IF P34_UzivatelPrihlaseny AND P34_Vizu.TL_PrihlasovOperatora_AKTIVNE THEN
		P34_Vizu.TL_PrihlasovOperatora_AKTIVNE:= FALSE;
	END_IF

	//************************************Zamknutie tlačítka editácia uživatelov***********************************************//
	IF P1_UrovenPrihlasenehoUzivatela < 100 THEN
		P1_Vizu.TL_Uzivatelia_ENABLE:= FALSE;
	ELSE
		P1_Vizu.TL_Uzivatelia_ENABLE:= TRUE;
	END_IF

END_PROGRAM

PROGRAM _EXIT
	(* Insert code here *)

END_PROGRAM
```

### Program Logical/Program/Linka/SafetyMapping_IO (IEC)

#### Main.st - Init, cyclic, exit code
```iecst
PROGRAM _INIT
	(* Insert code here *)

END_PROGRAM

PROGRAM _CYCLIC

	//********************************************Vstupy zo Safety do PLC****************************************************//
	Safety.STAV.P2_Bunka_VstupBariera_AKTIVNA:= Safety.Mapping_BYTE_IN[0].0;
	Safety.Mapping_BYTE_IN[0].1;
	Safety.STAV.P2_Bunka_Zamky_AKTIVNE:= Safety.Mapping_BYTE_IN[0].2;
	Safety.Mapping_BYTE_IN[0].3;
	Safety.STAV.P2_DvojrucOvl_TlacitkoCS_ODBLOK:= Safety.Mapping_BYTE_IN[0].4;
	Safety.Mapping_BYTE_IN[0].5;
	(*Safety.STAV.P2_DvojrucneOvladanie_AKTIVNE:= Safety.Mapping_BYTE_IN[0].6;*)
	Safety.Mapping_BYTE_IN[0].7;

	Safety.STAV.P1_Robot_TlacitkoCS_ODBLOK:= Safety.Mapping_BYTE_IN[1].0;
	Safety.Mapping_BYTE_IN[1].1;
	Safety.STAV.P1_Panel_TlacitkoCS_ODBLOK:= Safety.Mapping_BYTE_IN[1].2;
	Safety.Mapping_BYTE_IN[1].3;
	Safety.STAV.P1_VyblokovanieZamkov_AKTIVNE:= Safety.Mapping_BYTE_IN[1].4;
	Safety.Mapping_BYTE_IN[1].5;
	Safety.STAV.P1_Rozvadzac_TlacitkoCS_ODBLOK:= Safety.Mapping_BYTE_IN[1].6;
	Safety.Mapping_BYTE_IN[1].7;

	Safety.STAV.P1_Vytah_Muting_AKTIVNY:= Safety.Mapping_BYTE_IN[2].0;
	Safety.Mapping_BYTE_IN[2].1;
	Safety.STAV.P1_Bunka_Zamky_AKTIVNE:= Safety.Mapping_BYTE_IN[2].2;
	Safety.Mapping_BYTE_IN[2].3;
	Safety.STAV.P1_DeadMan_AKTIVNY:= Safety.Mapping_BYTE_IN[2].4;
	Safety.Mapping_BYTE_IN[2].5;
	Safety.STAV.P1_Vytah_Bariera_AKTIVNA:= Safety.Mapping_BYTE_IN[2].6;
	Safety.Mapping_BYTE_IN[2].7;

	Safety.STAV.P2_Robot_TlacitkoCS_ODBLOK:= Safety.Mapping_BYTE_IN[3].0;
	Safety.Mapping_BYTE_IN[3].1;
	Safety.STAV.P2_Panel_TlacitkoCS_ODBLOK:= Safety.Mapping_BYTE_IN[3].2;
	Safety.Mapping_BYTE_IN[3].3;
	Safety.STAV.P2_VyblokovanieZamkov_AKTIVNE:= Safety.Mapping_BYTE_IN[3].4;
	Safety.Mapping_BYTE_IN[3].5;
	Safety.STAV.P2_Rozvadzac_TlacitkoCS_ODBLOK:= Safety.Mapping_BYTE_IN[3].6;
	Safety.Mapping_BYTE_IN[3].7;

	Safety.STAV.P2_ZaklTesn_PojazdMuting_AKTIVNY:= Safety.Mapping_BYTE_IN[4].0;
	Safety.Mapping_BYTE_IN[4].1;
	Safety.STAV.P2_DeadMan_AKTIVNY:= Safety.Mapping_BYTE_IN[4].2;
	Safety.Mapping_BYTE_IN[4].3;
	Safety.STAV.P2_ZaklTesn_Bumper_AKTIVNY:= Safety.Mapping_BYTE_IN[4].4;
	Safety.Mapping_BYTE_IN[4].5;
	Safety.STAV.P2_ZaklTesn_Bariera_AKTIVNA:= Safety.Mapping_BYTE_IN[4].6;
	Safety.Mapping_BYTE_IN[4].7;

	Safety.Mapping_BYTE_IN[5].0;
	Safety.Mapping_BYTE_IN[5].1;
	Safety.STAV.P3_DeadMan_AKTIVNY:= Safety.Mapping_BYTE_IN[5].2;
	Safety.Mapping_BYTE_IN[5].3;
	Safety.STAV.P3_VyblokovanieZamkov_AKTIVNE:= Safety.Mapping_BYTE_IN[5].4;
	Safety.Mapping_BYTE_IN[5].5;
	Safety.STAV.P3_Rozvadzac_TlacitkoCS_ODBLOK:= Safety.Mapping_BYTE_IN[5].6;
	Safety.Mapping_BYTE_IN[5].7;

	Safety.STAV.P3_Bunka_Zamky_AKTIVNE:= Safety.Mapping_BYTE_IN[6].0;
	Safety.Mapping_BYTE_IN[6].1;
	Safety.STAV.P3_Bunka_VstupBariera_AKTIVNA:= Safety.Mapping_BYTE_IN[6].2;
	Safety.Mapping_BYTE_IN[6].3;
	Safety.STAV.P4_Bunka_VstupBariera_AKTIVNA:= Safety.Mapping_BYTE_IN[6].4;
	Safety.Mapping_BYTE_IN[6].5;
	Safety.Mapping_BYTE_IN[6].6;
	Safety.Mapping_BYTE_IN[6].7;

	Safety.STAV.P4_Panel_TlacitkoCS_ODBLOK:= Safety.Mapping_BYTE_IN[7].0;
	Safety.Mapping_BYTE_IN[7].1;
	Safety.STAV.P4_DeadMan_AKTIVNY:= Safety.Mapping_BYTE_IN[7].2;
	Safety.Mapping_BYTE_IN[7].3;
	Safety.STAV.P4_VyblokovanieZamkov_AKTIVNE:= Safety.Mapping_BYTE_IN[7].4;
	Safety.Mapping_BYTE_IN[7].5;
	Safety.STAV.P4_Rozvadzac_TlacitkoCS_ODBLOK:= Safety.Mapping_BYTE_IN[7].6;
	Safety.Mapping_BYTE_IN[7].7;

	Safety.STAV.P4_Bunka_Zamky_AKTIVNE:= Safety.Mapping_BYTE_IN[8].0;
	Safety.Mapping_BYTE_IN[8].1;
	Safety.STAV.P4_Vytah_Bariera_AKTIVNA:= Safety.Mapping_BYTE_IN[8].2;
	Safety.Mapping_BYTE_IN[8].3;
	Safety.STAV.P4_VystupBunky_VstupBar_AKTIVNA:= Safety.Mapping_BYTE_IN[8].4;
	Safety.Mapping_BYTE_IN[8].5;
	Safety.STAV.P4_VystupBunky_VystupBar_AKTIVNA:= Safety.Mapping_BYTE_IN[8].6;
	Safety.Mapping_BYTE_IN[8].7;

	Safety.STAV.P1_VstupBunky_VstupBar_AKTIVNA:= Safety.Mapping_BYTE_IN[9].0;
	Safety.Mapping_BYTE_IN[9].1;
	Safety.STAV.P1_VystupBunky_VstupBar_AKTIVNA:= Safety.Mapping_BYTE_IN[9].2;
	Safety.Mapping_BYTE_IN[9].3;
	Safety.STAV.P1_VstupBunky_VystupBar_AKTIVNA:= Safety.Mapping_BYTE_IN[9].4;
	Safety.Mapping_BYTE_IN[9].5;
	Safety.STAV.P1_VystupBunky_VystupBar_AKTIVNA:= Safety.Mapping_BYTE_IN[9].6;
	Safety.Mapping_BYTE_IN[9].7;

	Safety.STAV.P4_Vytah_Muting_AKTIVNY:= Safety.Mapping_BYTE_IN[13].0;
	Safety.Mapping_BYTE_IN[13].1;
	Safety.Mapping_BYTE_IN[13].2;
	Safety.Mapping_BYTE_IN[13].3;
	Safety.Mapping_BYTE_IN[13].4;
	Safety.Mapping_BYTE_IN[13].5;
	Safety.Mapping_BYTE_IN[13].6;
	Safety.Mapping_BYTE_IN[13].7;

	Safety.STAV.Linka_ZonaCS_AKTIVNA:= Safety.Mapping_BYTE_IN[16].0;
	Safety.STAV.P1_ZonaBunky_AKTIVNA:= Safety.Mapping_BYTE_IN[16].1;
	Safety.STAV.P1_ZonaVytahu_AKTIVNA:= Safety.Mapping_BYTE_IN[16].2;
	Safety.STAV.P2_ZonaBunky_AKTIVNA:= Safety.Mapping_BYTE_IN[16].3;
	Safety.STAV.P3_ZonaBunky_AKTIVNA:= Safety.Mapping_BYTE_IN[16].4;
	Safety.STAV.P3_ZonaHVtest_AKTIVNA:= Safety.Mapping_BYTE_IN[16].5;
	Safety.STAV.P4_ZonaBunky_AKTIVNA:= Safety.Mapping_BYTE_IN[16].6;
	Safety.STAV.P4_ZonaVytahu_AKTIVNA:= Safety.Mapping_BYTE_IN[16].7;

	IF Safety.STAV.P2_ZaklTesn_Bariera_AKTIVNA AND Safety.STAV.P2_ZaklTesn_PojazdMuting_AKTIVNY THEN
		Safety.STAV.P2_ZonaZakladacaZdvih_AKTIVNA:= TRUE;
	ELSE
		Safety.STAV.P2_ZonaZakladacaZdvih_AKTIVNA:= FALSE;
	END_IF

	IF Safety.Mapping_BYTE_IN[17].2 AND Safety.Mapping_BYTE_IN[17].3 THEN
		Safety.STAV.P2_ZonaMaticovacky_AKTIVNA:= TRUE;
	ELSE
		Safety.STAV.P2_ZonaMaticovacky_AKTIVNA:= FALSE;
	END_IF

	IF Safety.STAV.P2_ZaklTesn_Bumper_AKTIVNY THEN
		Safety.STAV.P2_ZonaZakladacaPojazd_AKTIVNA:= TRUE;
	ELSE
		Safety.STAV.P2_ZonaZakladacaPojazd_AKTIVNA:= FALSE;
	END_IF

	//***************************************************Výstupy pre Safety z PLC***********************************************************//
	Safety.Mapping_BYTE_OUT[0];

END_PROGRAM

PROGRAM _EXIT
	(* Insert code here *)

END_PROGRAM
```

### Program Logical/Program/Linka/StatistikaLinky (IEC)

#### Main.st - Init, cyclic, exit code
```iecst
PROGRAM _INIT

END_PROGRAM

PROGRAM _CYCLIC

	P1_Vytah_Taktime.IN.TaskovaTrieda_ms:= 4;
	P1_Skrutkovanie_Taktime.IN.TaskovaTrieda_ms:= 4;
	P2_ZakladanieTesnenia_Taktime.IN.TaskovaTrieda_ms:= 4;
	P2_Maticovacka_Taktime.IN.TaskovaTrieda_ms:= 4;
	P2_Skrutkovanie_Taktime.IN.TaskovaTrieda_ms:= 4;
	P2_Zvaranie_Taktime.IN.TaskovaTrieda_ms:= 4;
	P3_Skrutkovanie_Taktime.IN.TaskovaTrieda_ms:= 4;
	P3_HVtest_Taktime.IN.TaskovaTrieda_ms:= 4;
	P3_LeakageTestA_Taktime.IN.TaskovaTrieda_ms:= 4;
	P3_LeakageTestB_Taktime.IN.TaskovaTrieda_ms:= 4;
	P4_FinalTestA_Taktime.IN.TaskovaTrieda_ms:= 4;
	P4_FinalTestB_Taktime.IN.TaskovaTrieda_ms:= 4;
	P4_Etiketovanie_Taktime.IN.TaskovaTrieda_ms:= 4;
	P4_Vytah_Taktime.IN.TaskovaTrieda_ms:= 4;

	P1_Vytah_Taktime();
	P1_Skrutkovanie_Taktime();
	P2_ZakladanieTesnenia_Taktime();
	P2_Maticovacka_Taktime();
	P2_Skrutkovanie_Taktime();
	P2_Zvaranie_Taktime();
	P3_Skrutkovanie_Taktime();
	P3_HVtest_Taktime();
	P3_LeakageTestA_Taktime();
	P3_LeakageTestB_Taktime();
	P4_FinalTestA_Taktime();
	P4_FinalTestB_Taktime();
	P4_Etiketovanie_Taktime();
	P4_Vytah_Taktime();

END_PROGRAM

PROGRAM _EXIT
	(* Insert code here *)

END_PROGRAM
```

### Program Logical/Program/Pracovisko_1/P1_Main (IEC)

#### Main.st - Init, cyclic, exit code
```iecst
PROGRAM _INIT
	(* Insert code here *)

END_PROGRAM

PROGRAM _CYCLIC

	//Volanie podprogramov//
	ProfinetKomunikaciaKAM2;
	ProfinetKomunikaciaKAM3;
	ProfinetKomunikaciaKAM4;
	ProfinetKomunikaciaKAM5;
	ProfinetKomunikaciaKAM6;

	//**************************************Ukončenie cyklu pracoviska****************************************************//
	IF P1_Pracovisko.KoniecCyklu THEN
		IF P1_Dopravniky.Automat THEN
			P1_Dopravniky.KoniecCyklu:= TRUE;
		END_IF
		IF P1_SpodnyStoper.Automat THEN
			P1_SpodnyStoper.KoniecCyklu:= TRUE;
		END_IF
		IF P1_Vytah.Automat THEN
			P1_Vytah.KoniecCyklu:= TRUE;
		END_IF
		IF P1_StoperSrobovania.Automat THEN
			P1_StoperSrobovania.KoniecCyklu:= TRUE;
		END_IF
		IF P1_Srobovanie.Automat THEN
			P1_Srobovanie.KoniecCyklu:= TRUE;
		END_IF
		IF P1_Robot.Automat THEN
			P1_Robot.KoniecCyklu:= TRUE;
		END_IF
		IF P1_AkumulacnyStoper.Automat THEN
			P1_AkumulacnyStoper.KoniecCyklu:= TRUE;
		END_IF
		P1_Pracovisko.KoniecCyklu:= FALSE;
	END_IF

	//************************************Ukončenie cyklu pri poruche*****************************************//

	//ST1 - Výťah//
	IF P1_Pracovisko.STAV.Porucha_ST1 THEN
		IF P1_Vytah.Automat THEN
			P1_Vytah.Reset:= TRUE;
		END_IF
	END_IF

	//ST2 - Šrobovanie//
	IF P1_Pracovisko.STAV.Porucha_ST2 THEN
		IF P1_Dopravniky.Automat THEN
			P1_Dopravniky.KoniecCyklu:= TRUE;
		END_IF
		IF P1_SpodnyStoper.Automat THEN
			P1_SpodnyStoper.KoniecCyklu:= TRUE;
		END_IF
		IF P1_Srobovanie.Automat THEN
			P1_Srobovanie.Reset:= TRUE;
		END_IF
		IF P1_Robot.Automat THEN
			P1_Robot.KoniecCyklu:= TRUE;
		END_IF
		IF P1_AkumulacnyStoper.Automat THEN
			P1_AkumulacnyStoper.KoniecCyklu:= TRUE;
		END_IF
	END_IF

	//ST3 - Akumulačný stoper//
	IF P1_Pracovisko.STAV.Porucha_ST3 THEN
		IF P1_Dopravniky.Automat THEN
			P1_Dopravniky.KoniecCyklu:= TRUE;
		END_IF
		IF P1_SpodnyStoper.Automat THEN
			P1_SpodnyStoper.KoniecCyklu:= TRUE;
		END_IF
		IF P1_StoperSrobovania.Automat THEN
			P1_StoperSrobovania.KoniecCyklu:= TRUE;
		END_IF
		IF P1_Srobovanie.Automat THEN
			P1_Srobovanie.KoniecCyklu:= TRUE;
		END_IF
		IF P1_Robot.Automat THEN
			P1_Robot.KoniecCyklu:= TRUE;
		END_IF
		IF P1_AkumulacnyStoper.Automat THEN
			P1_AkumulacnyStoper.Reset:= TRUE;
		END_IF
	END_IF

	//*********************************Status prebieha ukončenie cyklu********************************************//
	IF P1_Vytah.KoniecCyklu OR
		P1_SpodnyStoper.KoniecCyklu OR
		P1_Dopravniky.KoniecCyklu OR
		P1_StoperSrobovania.KoniecCyklu OR
		P1_Srobovanie.KoniecCyklu OR
		P1_Robot.KoniecCyklu OR
		P1_AkumulacnyStoper.KoniecCyklu THEN
		P1_Pracovisko.STAV.UkoncenieCyklu_BUSY:= TRUE;
	ELSE
		P1_Pracovisko.STAV.UkoncenieCyklu_BUSY:= FALSE;
	END_IF

	//*******************************Resetovanie pracoviska po stlačení tlačítka Automat******************************************//
	IF P1_Vizu.TL_RezimAutomat THEN
		IF P1_Pracovisko.STAV.Manual THEN
			P1_Pracovisko.Reset:= TRUE;
		END_IF
		P1_Vizu.TL_RezimAutomat:= FALSE;
	END_IF

	//******************************************Resetovanie pracoviska************************************************************//
	IF P1_Pracovisko.Reset THEN
		P1_Vytah.Reset:= TRUE;
		P1_SpodnyStoper.Reset:= TRUE;
		P1_Dopravniky.Reset:= TRUE;
		P1_StoperSrobovania.Reset:= TRUE;
		P1_Srobovanie.Reset:= TRUE;
		P1_Robot.Reset:= TRUE;
		P1_AkumulacnyStoper.Reset:= TRUE;
		P1_Pracovisko.STAV.Porucha_ST1:= FALSE;
		P1_Pracovisko.STAV.Porucha_ST2:= FALSE;
		P1_Pracovisko.STAV.Porucha_ST3:= FALSE;
		P1_Pracovisko.Reset:= FALSE;
	END_IF

	//Prepnutie pracoviska do manualneho režimu//
	IF P1_Pracovisko.Manual THEN
		P1_Vytah.Manual:= TRUE;
		P1_SpodnyStoper.Manual:= TRUE;
		P1_Dopravniky.Manual:= TRUE;
		P1_StoperSrobovania.Manual:= TRUE;
		P1_Srobovanie.Manual:= TRUE;
		P1_Robot.Manual:= TRUE;
		P1_AkumulacnyStoper.Manual:= TRUE;
		P1_Pracovisko.Manual:= FALSE;
	END_IF

	//Spustenie pracoviska v automatickom režime//
	IF P1_Pracovisko.Automat THEN
		P1_SpodnyStoper.Automat:= TRUE;
		IF Safety.STAV.P1_ZonaVytahu_AKTIVNA AND P1_Pracovisko.STAV.HardwareVytahu_OK THEN
			P1_Vytah.Automat:= TRUE;
		END_IF
		IF Safety.STAV.P1_ZonaBunky_AKTIVNA AND P1_Pracovisko.STAV.HardwareBunky_OK THEN
			P1_Dopravniky.Automat:= TRUE;
			P1_StoperSrobovania.Automat:= TRUE;
			P1_Srobovanie.Automat:= TRUE;
			P1_Robot.Automat:= TRUE;
			P1_AkumulacnyStoper.Automat:= TRUE;
		END_IF
		P1_Pracovisko.Automat:= FALSE;
	END_IF

	//***************************************************Príznaky pracoviska******************************************************//
	//Príznak pracovisko stav AUTOMAT//
	IF P1_Vytah.Automat OR
		P1_SpodnyStoper.Automat OR
		P1_Dopravniky.Automat OR
		P1_StoperSrobovania.Automat OR
		P1_Srobovanie.Automat OR
		P1_Robot.Automat OR
		P1_AkumulacnyStoper.Automat THEN
		P1_Pracovisko.STAV.Automat:= TRUE;
	ELSE
		P1_Pracovisko.STAV.Automat:= FALSE;
	END_IF

	//Priznak pracovisko stav MANUAL//
	IF P1_Vytah.Manual OR
		P1_SpodnyStoper.Manual OR
		P1_Dopravniky.Manual OR
		P1_StoperSrobovania.Manual OR
		P1_Srobovanie.Manual OR
		P1_Robot.Manual OR
		P1_AkumulacnyStoper.Manual THEN
		P1_Pracovisko.STAV.Manual:= TRUE;
	ELSE
		P1_Pracovisko.STAV.Manual:= FALSE;
	END_IF

	//Príznak pracovisko stav PoINIT//
	IF P1_Vytah.STAV.PoINIT AND
		P1_SpodnyStoper.STAV.PoINIT AND
		P1_Dopravniky.STAV.PoINIT AND
		P1_StoperSrobovania.STAV.PoINIT AND
		P1_Srobovanie.STAV.PoINIT AND
		P1_Robot.STAV.PoINIT AND
		P1_AkumulacnyStoper.STAV.PoINIT THEN
		P1_Pracovisko.STAV.PoINIT:= TRUE;
	ELSE
		P1_Pracovisko.STAV.PoINIT:= FALSE;
	END_IF

	//Príznak pracovisko stav READY//
	IF SC_P1_Vytah.Step = 1 AND
		SC_P1_SpodnyStoper.Step = 1 AND
		SC_P1_Dopravniky.Step = 1 AND
		SC_P1_StoperSrobovania.Step = 1 AND
		SC_P1_Srobovanie.Step = 1 AND
		SC_P1_Robot.Step = 1 AND
		SC_P1_AkumulacnyStoper.Step = 1 THEN
		P1_Pracovisko.STAV.READY:= TRUE;
	ELSE
		P1_Pracovisko.STAV.READY:= FALSE;
	END_IF

	//Príznak pracovisko stav PORUCHA//
	IF P1_Pracovisko.STAV.Porucha_ST1 OR
		P1_Pracovisko.STAV.Porucha_ST2 OR
		P1_Pracovisko.STAV.Porucha_ST3 THEN
		P1_Pracovisko.STAV.PORUCHA:= TRUE;
	ELSE
		P1_Pracovisko.STAV.PORUCHA:= FALSE;
	END_IF

	//Priznak HW Vytahu OK//
	IF P1_Pracovisko.IN.TlakVzduchu_OK AND
		P1_Pracovisko.IN.ModulFesto_IO_KomOK AND
		P1_Pracovisko.IN.ModulWeidmuller_IO_KomOK AND
		P1_Pracovisko.IN.ServoZdvihuVytahu_KomOK AND
		P1_Pracovisko.IN.SmartKamera3_KomOK AND
		P1_Pracovisko.IN.SmartKamera5_KomOK AND
		P3_Pracovisko.IN.Kamery_ControlUnit_KomOK AND
		P1_Pracovisko.IN.VentilovyTerminal_KomOK THEN
		P1_Pracovisko.STAV.HardwareVytahu_OK:= TRUE;
	ELSE
		P1_Pracovisko.STAV.HardwareVytahu_OK:= FALSE;
	END_IF

	//Príznak HW Bunky OK//
	IF P1_Pracovisko.IN.TlakVzduchu_OK AND
		P1_Pracovisko.IN.ModulFesto_IO_KomOK AND
		P1_Pracovisko.IN.ModulWeidmuller_IO_KomOK AND
		P1_Pracovisko.IN.Robot_KomOK AND
		P1_Pracovisko.IN.ServoManipulatorOsX_KomOK AND
		P1_Pracovisko.IN.ServoManipulatorOsY_KomOK AND
		P1_Pracovisko.IN.ServoManipulatorOsZ_M4_KomOK AND
		P1_Pracovisko.IN.ServoManipulatorOsZ_M5_KomOK AND
		P1_Pracovisko.IN.Skrutkovacka_K30_KomOK AND
		P1_Pracovisko.IN.Skrutkovacka_M4_KomOK AND
		P1_Pracovisko.IN.Skrutkovacka_M5_KomOK AND
		P1_Srobovanie.IN.NapajanieSkrutkovackyK30_OK AND
		P1_Srobovanie.IN.NapajanieSkrutkovackyM4_OK AND
		P1_Srobovanie.IN.NapajanieSkrutkovackyM5_OK AND
		P1_Srobovanie.IN.NapajanieVibrolistyM4_OK AND
		P1_Srobovanie.IN.NapajanieVibrolistyM5_OK AND
		P1_Srobovanie.IN.NapajanieZasobnikaK30_OK AND
		P1_Srobovanie.IN.NapajanieZasobnikaM4_OK AND
		P1_Srobovanie.IN.NapajanieZasobnikaM5_OK AND
		P3_Pracovisko.IN.Kamery_ControlUnit_KomOK AND
		P1_Pracovisko.IN.VentilovyTerminal_KomOK THEN
		P1_Pracovisko.STAV.HardwareBunky_OK:= TRUE;
	ELSE
		P1_Pracovisko.STAV.HardwareBunky_OK:= FALSE;
	END_IF

	//Príznak skrutkovačky zasunuté//
	IF P1_Srobovanie.IN.Skrutkovacka_K30_ZASUNUTA AND P1_Srobovanie.PAR.ManipulOsZ_M4_AktualnaPozicia < 5 AND P1_Srobovanie.PAR.ManipulOsZ_M5_AktualnaPozicia < 5 THEN
		P1_Pracovisko.STAV.SkrutkovackyZasunute:= TRUE;
	ELSE
		P1_Pracovisko.STAV.SkrutkovackyZasunute:= FALSE;
	END_IF

	//*****************************Zapnutie osvetlenia pracoviska*********************************************************//
	(*P1_Pracovisko.OUT.OsvetlenieBunky_ON:= TRUE;*)
	P1_Vytah.OUT.OsvetlenieVytahu_ON:= TRUE;
	P1_Pracovisko.OUT.Osvetlenie_CAM5_ON:= TRUE;
	P1_Pracovisko.OUT.Osvetlenie_CAM6_ON:= TRUE;
	P1_Pracovisko.OUT.Srobovanie_BodoveOsvetlenie_ON:= TRUE;
	P1_Pracovisko.OUT.Srobovanie_OsvetleniePaletky_ON:= TRUE;

	//****************************************Ovládanie majáka***********************************************//
	//Zelené svetlo//
	IF P1_Pracovisko.STAV.Automat THEN
		P1_Pracovisko.OUT.Majak_ZeleneSvetlo_ON:= TRUE;
	ELSIF P1_Pracovisko.STAV.Manual THEN
		P1_Pracovisko.OUT.Majak_ZeleneSvetlo_ON:= Blikac500ms;
	ELSE
		P1_Pracovisko.OUT.Majak_ZeleneSvetlo_ON:= FALSE;
	END_IF

	//Oranžové svetlo//
	IF P1_Pracovisko.STAV.Automat AND NOT P1_Pracovisko.STAV.PoINIT THEN
		P1_Pracovisko.OUT.Majak_OranzoveSvetlo_ON:= TRUE;
	ELSE
		P1_Pracovisko.OUT.Majak_OranzoveSvetlo_ON:= FALSE;
	END_IF

	//Červené svetlo//
	IF NOT Safety.STAV.Linka_ZonaCS_AKTIVNA THEN
		P1_Pracovisko.OUT.Majak_CerveneSvetlo_ON:= TRUE;
	ELSIF P1_Pracovisko.STAV.Porucha_ST1 THEN
		P1_Pracovisko.OUT.Majak_CerveneSvetlo_ON:= TRUE;
	ELSIF P1_Pracovisko.STAV.Porucha_ST2 THEN
		P1_Pracovisko.OUT.Majak_CerveneSvetlo_ON:= TRUE;
	ELSIF P1_Pracovisko.STAV.Porucha_ST3 THEN
		P1_Pracovisko.OUT.Majak_CerveneSvetlo_ON:= TRUE;
	ELSE
		P1_Pracovisko.OUT.Majak_CerveneSvetlo_ON:= FALSE;
	END_IF

	//Zvuková signalizácia//
	//	IF EDGEPOS(P1_Pracovisko.STAV.Porucha_ST1) THEN
	//		P1_Pracovisko.OUT.Majak_Hukacka_ON:= Blikac500ms;
	//	ELSIF EDGEPOS(P1_Pracovisko.STAV.Porucha_ST2) THEN
	//		P1_Pracovisko.OUT.Majak_Hukacka_ON:= Blikac500ms;
	//	ELSIF EDGEPOS(P1_Pracovisko.STAV.Porucha_ST3) THEN
	//		P1_Pracovisko.OUT.Majak_Hukacka_ON:= Blikac500ms;
	//	END_IF

END_PROGRAM

PROGRAM _EXIT
		(* Insert code here *)

END_PROGRAM
```

#### Variables.var - Local variables
```iecst
VAR
	Convert_0 : UsintToUint := (0);
	Convert_1 : UsintToUint := (0);
	Convert_2 : UsintToUint := (0);
	Convert_3 : UsintToUint := (0);
	Convert_4 : UsintToUint := (0);
END_VAR
```

#### ProfinetKomunikaciaKAM3.st
```iecst
ACTION ProfinetKomunikaciaKAM3:

	//Smart kamera//
	CAM3.STAV.READY:= P1_Pracovisko.IN.SmartKamera3_KomOK;

	//Vstupy pre kameru//
	CAM3.Profinet_PLC_OUTPUTS[0].0:= CAM3.CMD.Triger;

	//Výstupy z kamery//
	CAM3.STAV.SWITCH:= CAM3.Profinet_PLC_INPUTS[12].0;

	//Výsledky kamery//
	CAM3.RESULT.Paletka.CitanieQRkodu_DPS_OK:= CAM3.Profinet_PLC_INPUTS[0].0;

	//Prečítaný QR kód DPS//
	IF EDGE(CAM3.STAV.SWITCH) THEN
		brsstrcpy(ADR(CAM3.RESULT.Paletka.PrecitanyQRkod_DPS),ADR(CAM3.Profinet_QRkod_Znaky));
	END_IF

	//Stav výsledky READY//
	IF EDGE(CAM3.STAV.SWITCH)THEN
		CAM3.STAV.Results_READY:= TRUE;
	END_IF

	//Run counter kamery//
	Convert_0.IN_Byte0:= CAM3.STAV.RunCounter_Byte1;
	Convert_0.IN_Byte1:= CAM3.STAV.RunCounter_Byte0;

	CAM3.STAV.RunCounter:= Convert_0.OUT_UINT;
	Convert_0();

END_ACTION
```

#### ProfinetKomunikaciaKAM2.st
```iecst
ACTION ProfinetKomunikaciaKAM2:
	//Control unit CAM1//

	//Vstupy pre kameru//
	CAM2.Profinet_PLC_OUTPUTS[0].3:= CAM2.CMD.Triger;

	//Výstupy z kamery//
	CAM2.STAV.READY:= CAM2.Profinet_PLC_INPUTS[0].0;
	CAM2.STAV.SWITCH:= CAM2.Profinet_PLC_INPUTS[0].1;
    CAM2.STAV.BUSY:= CAM2.Profinet_PLC_INPUTS[0].2;
    CAM2.STAV.Command_AKCEPTOVANY:= CAM2.Profinet_PLC_INPUTS[0].3;
    CAM2.STAV.Command_READY:= CAM2.Profinet_PLC_INPUTS[0].4;
    CAM2.STAV.Command_ERROR:= CAM2.Profinet_PLC_INPUTS[0].5;

	//Výsledky kamery//
	CAM2.RESULT.Paletka.Pritom_PowerCP_4F:= CAM2.Profinet_PLC_INPUTS[2].0;
	CAM2.RESULT.Paletka.Pritom_PowerCP_5F:= CAM2.Profinet_PLC_INPUTS[2].1;
	CAM2.RESULT.Paletka.Pritom_PowerCP_5H:= CAM2.Profinet_PLC_INPUTS[2].2;
	CAM2.RESULT.Paletka.Pritomn_Skeletonu_5H:= CAM2.Profinet_PLC_INPUTS[2].3;
	CAM2.RESULT.Paletka.Pritomn_Skeletonu_4F5F:= CAM2.Profinet_PLC_INPUTS[2].4;
	CAM2.RESULT.Paletka.Pritom_Busbarov_Spodne_5H:= CAM2.Profinet_PLC_INPUTS[2].5;
	CAM2.RESULT.Paletka.Pritom_Foamu_Lavy_4F5F:= CAM2.Profinet_PLC_INPUTS[2].6;
	CAM2.RESULT.Paletka.Pritom_Foamu_Pravy_4F5F:= CAM2.Profinet_PLC_INPUTS[2].7;
	CAM2.RESULT.Paletka.Pritom_Busbaru_Spodny_4F:= CAM2.Profinet_PLC_INPUTS[3].0;
	CAM2.RESULT.Paletka.Pritom_Busbaru_Spodny_5F:= CAM2.Profinet_PLC_INPUTS[3].1;
	CAM2.RESULT.Paletka.Pritom_DPS_4F5F:= CAM2.Profinet_PLC_INPUTS[3].2;

	//Stav výsledky READY//
	IF EDGE(CAM2.STAV.SWITCH)THEN
		CAM2.STAV.Results_READY:= TRUE;
		CAM2_PocetFotiek:= CAM2_PocetFotiek + 1;
	END_IF

	//Vymazanie adresára kamery//
	IF EDGEPOS(CAM2_PocetFotiek > 50) THEN
		FTP_CAM2.CMD.VymazFotku:= TRUE;
		FTP_CAM2.STATUS.VymazanieAdresaraKamery_BUSY:= TRUE;
	END_IF

	IF (FTP_CAM2.STATUS.KomunikaciaUkoncena OR FTP_CAM2.STATUS.KomunikaciaError) AND FTP_CAM2.STATUS.VymazanieAdresaraKamery_BUSY THEN
		FTP_CAM2.CMD.VymazFotku:= FALSE;
		FTP_CAM2.STATUS.VymazanieAdresaraKamery_BUSY:= FALSE;
	END_IF

	//Run counter kamery//
	Convert_1.IN_Byte0:= CAM2.STAV.RunCounter_Byte1;
	Convert_1.IN_Byte1:= CAM2.STAV.RunCounter_Byte0;

	CAM2.STAV.RunCounter:= Convert_1.OUT_UINT;
	Convert_1();

END_ACTION
```

#### ProfinetKomunikaciaKAM4.st
```iecst
ACTION ProfinetKomunikaciaKAM4:
	//Control unit CAM2//

	//Vstupy pre kameru//
	CAM4.Profinet_PLC_OUTPUTS[0].3:= CAM4.CMD.Triger;

	//Výstupy z kamery//
	CAM4.STAV.READY:= CAM4.Profinet_PLC_INPUTS[0].0;
	CAM4.STAV.SWITCH:= CAM4.Profinet_PLC_INPUTS[0].1;
    CAM4.STAV.BUSY:= CAM4.Profinet_PLC_INPUTS[0].2;
    CAM4.STAV.Command_AKCEPTOVANY:= CAM4.Profinet_PLC_INPUTS[0].3;
    CAM4.STAV.Command_READY:= CAM4.Profinet_PLC_INPUTS[0].4;
    CAM4.STAV.Command_ERROR:= CAM4.Profinet_PLC_INPUTS[0].5;

	//Výsledky kamery//
	CAM4.RESULT.Paletka.Pritomn_Pinu1_KrytDPS_4F5F:= CAM4.Profinet_PLC_INPUTS[2].0;
	CAM4.RESULT.Paletka.Pritomn_Pinu2_KrytDPS_4F5F:= CAM4.Profinet_PLC_INPUTS[2].1;
	CAM4.RESULT.Paletka.Pritomn_Pinu3_KrytDPS_4F5F:= CAM4.Profinet_PLC_INPUTS[2].2;
	CAM4.RESULT.Paletka.Pritomn_Pinu4_KrytDPS_4F5F:= CAM4.Profinet_PLC_INPUTS[2].3;
	CAM4.RESULT.Paletka.Pritomn_Pinu5_KrytDPS_4F5F:= CAM4.Profinet_PLC_INPUTS[2].4;
	CAM4.RESULT.Paletka.Pritomn_Pinu6_KrytDPS_4F5F:= CAM4.Profinet_PLC_INPUTS[2].5;
	CAM4.RESULT.Paletka.Pritom_DPS_4F5F:= CAM4.Profinet_PLC_INPUTS[2].6;

	//Stav výsledky READY//
	IF EDGE(CAM4.STAV.SWITCH)THEN
		CAM4.STAV.Results_READY:= TRUE;
		CAM4_PocetFotiek:= CAM4_PocetFotiek + 1;
	END_IF

	//Vymazanie adresára kamery//
	IF EDGEPOS(CAM4_PocetFotiek > 50) THEN
		FTP_CAM4.CMD.VymazFotku:= TRUE;
		FTP_CAM4.STATUS.VymazanieAdresaraKamery_BUSY:= TRUE;
	END_IF

	IF (FTP_CAM4.STATUS.KomunikaciaUkoncena OR FTP_CAM4.STATUS.KomunikaciaError) AND FTP_CAM4.STATUS.VymazanieAdresaraKamery_BUSY THEN
		FTP_CAM4.CMD.VymazFotku:= FALSE;
		FTP_CAM4.STATUS.VymazanieAdresaraKamery_BUSY:= FALSE;
	END_IF

	//Run counter kamery//
	Convert_2.IN_Byte0:= CAM4.STAV.RunCounter_Byte1;
	Convert_2.IN_Byte1:= CAM4.STAV.RunCounter_Byte0;

	CAM4.STAV.RunCounter:= Convert_2.OUT_UINT;
	Convert_2();

END_ACTION
```

#### ProfinetKomunikaciaKAM6.st
```iecst
ACTION ProfinetKomunikaciaKAM6:
	//Control unit CAM3//

	//Vstupy pre kameru//
	CAM6.Profinet_PLC_OUTPUTS[0].3:= CAM6.CMD.Triger;

	//Výstupy z kamery//
	CAM6.STAV.READY:= CAM6.Profinet_PLC_INPUTS[0].0;
	CAM6.STAV.SWITCH:= CAM6.Profinet_PLC_INPUTS[0].1;
    CAM6.STAV.BUSY:= CAM6.Profinet_PLC_INPUTS[0].2;
    CAM6.STAV.Command_AKCEPTOVANY:= CAM6.Profinet_PLC_INPUTS[0].3;
    CAM6.STAV.Command_READY:= CAM6.Profinet_PLC_INPUTS[0].4;
    CAM6.STAV.Command_ERROR:= CAM6.Profinet_PLC_INPUTS[0].5;

	//Výsledky kamery//
	CAM6.RESULT.Paletka.Pritom_PowerCP_5H:= CAM6.Profinet_PLC_INPUTS[2].0;
	CAM6.RESULT.Paletka.Pritom_SpodnychBusbarov_5H:= CAM6.Profinet_PLC_INPUTS[2].1;
	CAM6.RESULT.Paletka.Pritom_PowerCP_4F:= CAM6.Profinet_PLC_INPUTS[2].2;
	CAM6.RESULT.Paletka.Pritom_PowerCP_5F:= CAM6.Profinet_PLC_INPUTS[2].3;
	CAM6.RESULT.Paletka.Pritom_LavyFoam_4F5F:= CAM6.Profinet_PLC_INPUTS[2].4;
	CAM6.RESULT.Paletka.Pritom_PravyFoam_4F5F:= CAM6.Profinet_PLC_INPUTS[2].5;
	CAM6.RESULT.Paletka.Pritom_DPS_45F:= CAM6.Profinet_PLC_INPUTS[2].6;
	CAM6.RESULT.Paletka.Pritom_SpodnyBusbar_4F:= CAM6.Profinet_PLC_INPUTS[2].7;

	CAM6.RESULT.Paletka.Pritom_SpodnyBusbar_5F:= CAM6.Profinet_PLC_INPUTS[3].0;
	CAM6.RESULT.PowerCP.Nepritom_LavyFoam_4F5F:= CAM6.Profinet_PLC_INPUTS[3].1;
	CAM6.RESULT.PowerCP.Nepritom_PravyFoam_4F5F:= CAM6.Profinet_PLC_INPUTS[3].2;
	CAM6.RESULT.PowerCP.Pritom_LavejSkrutkyK30:= CAM6.Profinet_PLC_INPUTS[3].3;
	CAM6.RESULT.PowerCP.Pritom_PravejSkrutkyK30:= CAM6.Profinet_PLC_INPUTS[3].4;

	//Stav výsledky READY//
	IF EDGE(CAM6.STAV.SWITCH)THEN
		CAM6.STAV.Results_READY:= TRUE;
		CAM6_PocetFotiek:= CAM6_PocetFotiek + 1;
	END_IF

	//Vymazanie adresára kamery//
	IF EDGEPOS(CAM6_PocetFotiek > 50) THEN
		FTP_CAM6.CMD.VymazFotku:= TRUE;
		FTP_CAM6.STATUS.VymazanieAdresaraKamery_BUSY:= TRUE;
	END_IF

	IF (FTP_CAM6.STATUS.KomunikaciaUkoncena OR FTP_CAM6.STATUS.KomunikaciaError) AND FTP_CAM6.STATUS.VymazanieAdresaraKamery_BUSY THEN
		FTP_CAM6.CMD.VymazFotku:= FALSE;
		FTP_CAM6.STATUS.VymazanieAdresaraKamery_BUSY:= FALSE;
	END_IF

	//Run counter kamery//
	Convert_3.IN_Byte0:= CAM6.STAV.RunCounter_Byte1;
	Convert_3.IN_Byte1:= CAM6.STAV.RunCounter_Byte0;

	CAM6.STAV.RunCounter:= Convert_3.OUT_UINT;
	Convert_3();

END_ACTION
```

#### ProfinetKomunikaciaKAM5.st
```iecst
ACTION ProfinetKomunikaciaKAM5:
	//Smart kamera//

	CAM5.STAV.READY:= P1_Pracovisko.IN.SmartKamera5_KomOK;

	//Vstupy pre kameru//
	CAM5.Profinet_PLC_OUTPUTS[0].0:= CAM5.CMD.Triger;

	//Výstupy z kamery//
	CAM5.STAV.SWITCH:= CAM5.Profinet_PLC_INPUTS[12].0;

	//Výsledky kamery//
	CAM5.RESULT.PowerCP.CitanieQRkodu_PowerCP_OK:= CAM5.Profinet_PLC_INPUTS[0].0;

	//Prečítaný QR kód DPS//
	IF EDGE(CAM5.STAV.SWITCH) THEN
		brsstrcpy(ADR(CAM5.RESULT.PowerCP.PrecitanyQRkod_PowerCP),ADR(CAM5.Profinet_QRkod_Znaky));
	END_IF

	//Stav výsledky READY//
	IF EDGE(CAM5.STAV.SWITCH)THEN
		CAM5.STAV.Results_READY:= TRUE;
	END_IF

	//Run counter kamery//
	Convert_4.IN_Byte0:= CAM5.STAV.RunCounter_Byte1;
	Convert_4.IN_Byte1:= CAM5.STAV.RunCounter_Byte0;

	CAM5.STAV.RunCounter:= Convert_4.OUT_UINT;
	Convert_4();

END_ACTION
```

### Program Logical/Program/Pracovisko_1/P1_Dopravniky (IEC)

#### Main.st - Init, cyclic, exit code
```iecst
PROGRAM _INIT
	(* Insert code here *)

END_PROGRAM

PROGRAM _CYCLIC

	//Volanie funkcie SequenceControl//
	SequenceControl(SC:= SC_P1_Dopravniky);

	//Reset sekcie //
	IF P1_Dopravniky.Reset THEN
		SC_P1_Dopravniky.Step:= 0;
		P1_Dopravniky.Reset:= FALSE;
	ELSIF NOT Safety.STAV.Linka_ZonaCS_AKTIVNA THEN
		SC_P1_Dopravniky.Step:= 0;
	END_IF

	CASE SC_P1_Dopravniky.Step OF

		0:
			SC_P1_Dopravniky.StepName:='0 - Nulovanie';
			P1_Dopravniky.Automat:= FALSE;
			P1_Dopravniky.KoniecCyklu:= FALSE;
			P1_Dopravniky.Manual:= FALSE;
			P1_Dopravniky.STAV.PoINIT:= FALSE;
			P1_Dopravniky.OUT.DopravnikBunky_ON:= FALSE;
			P1_Dopravniky.OUT.VratnyDopravnik_ON:= FALSE;

			IF Safety.STAV.Linka_ZonaCS_AKTIVNA AND NOT P1_Pracovisko.STAV.PORUCHA AND P1_Pracovisko.STAV.HardwareBunky_OK THEN
				SC_P1_Dopravniky.ResetStep:= TRUE;
				SC_P1_Dopravniky.Step:= 1;
			END_IF

		1:
			SC_P1_Dopravniky.StepName:='1 - Cakam na spustenie vyroby';
			P1_Dopravniky.KoniecCyklu:= FALSE;
			IF P1_Dopravniky.Automat THEN
				SC_P1_Dopravniky.Step:= 2;
			ELSIF P1_Dopravniky.Manual THEN
				SC_P1_Dopravniky.Step:= 700;
			END_IF

			//********************************************************Inicializácia****************************************************************************//

		2:
			SC_P1_Dopravniky.StepName:='2 - Inicializacia - cakam na spustenie inicializacie';
			SC_P1_Dopravniky.IdleTime.PT:= T#1s;
			SC_P1_Dopravniky.AlarmTime.PT:= T#5s;

			IF P1_Pracovisko.STAV.SkrutkovackyZasunute AND P1_Robot.STAV.PoINIT THEN
				SC_P1_Dopravniky.IdleTime.IN:= TRUE;
			ELSE
				SC_P1_Dopravniky.IdleTime.IN:= FALSE;
			END_IF

			IF SC_P1_Dopravniky.IdleTime.Q THEN
				SC_P1_Dopravniky.ResetStep:= TRUE;
				SC_P1_Dopravniky.Step:= 3;
			END_IF

		3:
			SC_P1_Dopravniky.StepName:='3 - Inicializacia - inicializacia tlmenia stoprov';
			SC_P1_Dopravniky.IdleTime.PT:= T#1s;
			SC_P1_Dopravniky.AlarmTime.PT:= T#5s;

			IF P1_StoperSrobovania.RFID_hlava.PritomnostPaletky AND
				P1_AkumulacnyStoper.IN.PritomnostPaletky AND
				P1_SpodnyStoper.IN.PritomnostPaletky THEN
				SC_P1_Dopravniky.ResetStep:= TRUE;
				SC_P1_Dopravniky.Step:= 5;
			ELSE
				IF NOT P1_StoperSrobovania.RFID_hlava.PritomnostPaletky AND P1_StoperSrobovania.IN.Centrovanie_ZASUNUTE THEN
					P1_StoperSrobovania.OUT.ZasunStoper:= TRUE;
				END_IF
				IF NOT P1_AkumulacnyStoper.IN.PritomnostPaletky THEN
					P1_AkumulacnyStoper.OUT.ZasunStoper:= TRUE;
				END_IF
				IF NOT P1_SpodnyStoper.IN.PritomnostPaletky THEN
					P1_SpodnyStoper.OUT.ZasunStoper:= TRUE;
				END_IF
				SC_P1_Dopravniky.IdleTime.IN:= TRUE;
			END_IF

			IF SC_P1_Dopravniky.IdleTime.Q THEN
				P1_StoperSrobovania.OUT.ZasunStoper:= FALSE;
				P1_AkumulacnyStoper.OUT.ZasunStoper:= FALSE;
				P1_SpodnyStoper.OUT.ZasunStoper:= FALSE;
				SC_P1_Dopravniky.ResetStep:= TRUE;
				SC_P1_Dopravniky.Step:= 5;
			END_IF

		5:
			SC_P2_Dopravniky.StepName:='5 - Inicializacia - ukoncenie inicializacie';
			SC_P2_Dopravniky.IdleTime.PT:= T#5s;
			SC_P2_Dopravniky.AlarmTime.PT:= T#5s;

			P1_Dopravniky.OUT.DopravnikBunky_ON:= TRUE;
			P1_Dopravniky.OUT.VratnyDopravnik_ON:= TRUE;
			SC_P1_Dopravniky.IdleTime.IN:= TRUE;

			IF SC_P1_Dopravniky.IdleTime.Q THEN
				P1_Dopravniky.STAV.PoINIT:= TRUE;
				SC_P1_Dopravniky.ResetStep:= TRUE;
				SC_P1_Dopravniky.Step:= 100;
			END_IF

			//********************************************************Automatický režim****************************************************************************//

		100:
			SC_P1_Dopravniky.StepName:='100 - Automaticky Rezim - cakam na vypnutie dopravnikou';
			SC_P1_Dopravniky.IdleTime.PT:= T#200ms;
			SC_P1_Dopravniky.AlarmTime.PT:= T#5s;

			IF P1_Dopravniky.KoniecCyklu AND
				NOT P1_Vytah.STAV.PrebiehaVyvezeniePaletky AND
				NOT P1_StoperSrobovania.Automat AND
				NOT P1_AkumulacnyStoper.Automat AND
				NOT P1_SpodnyStoper.Automat THEN
				SC_P1_Dopravniky.ResetStep:= TRUE;
				SC_P1_Dopravniky.Step:= 0;
			END_IF

			//*******************************************************Manuálny režim*******************************************************************************//
		700:
			SC_P1_Dopravniky.StepName:='700 - Manualny Rezim';
			SC_P1_Dopravniky.IdleTime.PT:= T#8s;
			SC_P1_Dopravniky.AlarmTime.PT:= T#5s;

	END_CASE

END_PROGRAM

PROGRAM _EXIT
	(* Insert code here *)

END_PROGRAM
```

### Program Logical/Program/Pracovisko_1/P1_SpodnyStoper (IEC)

#### Main.st - Init, cyclic, exit code
```iecst
PROGRAM _INIT
	(* Insert code here *)

END_PROGRAM

PROGRAM _CYCLIC

	//Volanie funkcie SequenceControl//
	SequenceControl(SC:= SC_P1_SpodnyStoper);

	//Reset sekcie //
	IF P1_SpodnyStoper.Reset THEN
		SC_P1_SpodnyStoper.Step:= 0;
		P1_SpodnyStoper.Reset:= FALSE;
	ELSIF NOT Safety.STAV.Linka_ZonaCS_AKTIVNA THEN
		SC_P1_SpodnyStoper.Step:= 0;
	END_IF

	CASE SC_P1_SpodnyStoper.Step OF

		0:
			SC_P1_SpodnyStoper.StepName:='0 - Nulovanie';
			P1_SpodnyStoper.Automat:= FALSE;
			P1_SpodnyStoper.KoniecCyklu:= FALSE;
			P1_SpodnyStoper.Manual:= FALSE;
			P1_SpodnyStoper.STAV.PoINIT:= FALSE;
			P1_SpodnyStoper.STAV.PrebiehaVyvezeniePaletky:= FALSE;
			P1_SpodnyStoper.OUT.ZasunStoper:= FALSE;

			IF Safety.STAV.Linka_ZonaCS_AKTIVNA AND P1_Pracovisko.STAV.HardwareBunky_OK THEN
				SC_P1_SpodnyStoper.ResetStep:= TRUE;
				SC_P1_SpodnyStoper.Step:= 1;
			END_IF

		1:
			SC_P1_SpodnyStoper.StepName:='1 - Cakam na spustenie vyroby';
			P1_SpodnyStoper.KoniecCyklu:= FALSE;
			IF P1_SpodnyStoper.Automat THEN
				SC_P1_SpodnyStoper.Step:= 2;
			ELSIF P1_SpodnyStoper.Manual THEN
				SC_P1_SpodnyStoper.Step:= 700;
			END_IF

			//********************************************************Inicializácia****************************************************************************//
		2:
			SC_P1_SpodnyStoper.StepName:='2 - Inicializacia - cakam na spustenie inicializacie';
			SC_P1_SpodnyStoper.IdleTime.PT:= T#4s;
			SC_P1_SpodnyStoper.AlarmTime.PT:= T#5s;

			IF P1_Dopravniky.STAV.PoINIT THEN
				SC_P1_SpodnyStoper.ResetStep:= TRUE;
				SC_P1_SpodnyStoper.Step:= 3;
			END_IF

		3:
			SC_P1_SpodnyStoper.StepName:='3 - Inicializacia - hladanie paletky';
			SC_P1_SpodnyStoper.IdleTime.PT:= T#5s;
			SC_P1_SpodnyStoper.AlarmTime.PT:= T#5s;
			SC_P1_SpodnyStoper.IdleTime.IN:= TRUE;

			IF P1_SpodnyStoper.IN.PritomnostPaletky THEN
				P1_SpodnyStoper.STAV.PoINIT:= TRUE;
				SC_P1_SpodnyStoper.ResetStep:= TRUE;
				SC_P1_SpodnyStoper.Step:= 101;
			ELSIF SC_P1_SpodnyStoper.IdleTime.Q THEN
				P1_SpodnyStoper.STAV.PoINIT:= TRUE;
				SC_P1_SpodnyStoper.ResetStep:= TRUE;
				SC_P1_SpodnyStoper.Step:= 100;
			END_IF

			//********************************************************Automatický režim****************************************************************************//
		100:
			SC_P1_SpodnyStoper.StepName:='100 - Automaticky Rezim - cakam na príchod paletky na stoper';
			SC_P1_SpodnyStoper.IdleTime.PT:= T#200ms;
			SC_P1_SpodnyStoper.AlarmTime.PT:= T#5s;

			SC_P1_SpodnyStoper.IdleTime.IN:= P1_SpodnyStoper.IN.PritomnostPaletky;

			IF P1_SpodnyStoper.KoniecCyklu AND SC_P1_Vytah.Step <> 103 AND SC_P1_Vytah.Step <> 105 THEN
				SC_P1_SpodnyStoper.ResetStep:= TRUE;
				SC_P1_SpodnyStoper.Step:= 0;
			ELSIF SC_P1_SpodnyStoper.IdleTime.Q THEN
				SC_P1_SpodnyStoper.ResetStep:= TRUE;
				SC_P1_SpodnyStoper.Step:= 101;
			END_IF

		101:
			SC_P1_SpodnyStoper.StepName:='101 - Automaticky Rezim - cakam na vyvezenie paletky na dopravnik vytahu';
			SC_P1_SpodnyStoper.IdleTime.PT:= T#200ms;
			SC_P1_SpodnyStoper.AlarmTime.PT:= T#5s;

			IF P1_SpodnyStoper.KoniecCyklu AND SC_P1_Vytah.Step <> 103 AND SC_P1_Vytah.Step <> 105 THEN
				SC_P1_SpodnyStoper.ResetStep:= TRUE;
				SC_P1_SpodnyStoper.Step:= 0;
			ELSIF SC_P1_Vytah.Step = 105 AND NOT P1_Vytah.RFID_hlava.PritomnostPaletky THEN
				SC_P1_SpodnyStoper.ResetStep:= TRUE;
				SC_P1_SpodnyStoper.Step:= 105;
			ELSIF NOT P1_SpodnyStoper.IN.PritomnostPaletky THEN
				SC_P1_SpodnyStoper.ResetStep:= TRUE;
				SC_P1_SpodnyStoper.Step:= 100;
			END_IF

		105:
			SC_P1_SpodnyStoper.StepName:='105 - Automaticky Rezim - vyvazam paletku na dopravnik vytahu';
			SC_P1_SpodnyStoper.IdleTime.PT:= T#200ms;
			SC_P1_SpodnyStoper.AlarmTime.PT:= T#10s;

			SC_P1_SpodnyStoper.AlarmTime.IN:= P1_SpodnyStoper.IN.PritomnostPaletky;

			IF NOT SC_P1_SpodnyStoper.Switch1 THEN
				P1_SpodnyStoper.OUT.ZasunStoper:= TRUE;
				P1_SpodnyStoper.STAV.PrebiehaVyvezeniePaletky:= TRUE;
				SC_P1_SpodnyStoper.Switch1:= TRUE;
			END_IF

			IF NOT P1_SpodnyStoper.IN.PritomnostPaletky THEN
				P1_SpodnyStoper.OUT.ZasunStoper:= FALSE;
				SC_P1_SpodnyStoper.ResetStep:= TRUE;
				SC_P1_SpodnyStoper.Step:= 108;
			ELSIF SC_P1_SpodnyStoper.AlarmTime.Q THEN
				P1_Alarmy[163]:= TRUE;
				P1_Pracovisko.STAV.Porucha_ST1:= TRUE;
				SC_P1_SpodnyStoper.ResetStep:= TRUE;
				SC_P1_SpodnyStoper.Step:= 0;
			END_IF

		108:
			SC_P1_SpodnyStoper.StepName:='108 - Automaticky Rezim - cakam na prichod paletky na dopravnik vytahu';
			SC_P1_SpodnyStoper.IdleTime.PT:= T#200ms;
			SC_P1_SpodnyStoper.AlarmTime.PT:= T#10s;

			IF P1_Vytah.RFID_hlava.PritomnostPaletky THEN
				P1_SpodnyStoper.STAV.PrebiehaVyvezeniePaletky:= FALSE;
				SC_P1_SpodnyStoper.ResetStep:= TRUE;
				SC_P1_SpodnyStoper.Step:= 100;
			END_IF

			//*******************************************************Manuálny režim*******************************************************************************//
		700:
			SC_P1_SpodnyStoper.StepName:='700 - Manualny Rezim';
			SC_P1_SpodnyStoper.IdleTime.PT:= T#8s;
			SC_P1_SpodnyStoper.AlarmTime.PT:= T#5s;

	END_CASE

END_PROGRAM

PROGRAM _EXIT
	(* Insert code here *)

END_PROGRAM
```

### Program Logical/Program/Pracovisko_1/P1_Vytah (IEC)
